LIN {X 0,Y 125.805,Z 374.565,A -85,B 0,C 180,E1 -26043.072,E2 -26043.072} C_VEL
LIN {X 0,Y 129.803,Z 368.331,A -85,B 0,C 180,E1 -26046.553,E2 -26046.553} C_VEL
LIN {X 0,Y 133.449,Z 362.382,A -85,B 0,C 180,E1 -26049.195,E2 -26049.195} C_VEL
LIN {X 0,Y 137.426,Z 355.46,A -85,B 0,C 180,E1 -26051.668,E2 -26051.668} C_VEL
LIN {X 0,Y 141.639,Z 347.287,A -85,B 0,C 180,E1 -26054,E2 -26054} C_VEL
LIN {X 0,Y 145.555,Z 338.782,A -85,B 0,C 180,E1 -26055.907,E2 -26055.907} C_VEL
LIN {X 0,Y 149.029,Z 330.073,A -85,B 0,C 180,E1 -26057.464,E2 -26057.464} C_VEL
LIN {X 0,Y 152.312,Z 320.32,A -85,B 0,C 180,E1 -26058.823,E2 -26058.823} C_VEL
LIN {X 0,Y 155.098,Z 310.244,A -85,B 0,C 180,E1 -26059.876,E2 -26059.876} C_VEL
LIN {X 0,Y 157.131,Z 300.522,A -85,B 0,C 180,E1 -26060.648,E2 -26060.648} C_VEL
LIN {X 0,Y 158.62,Z 290.465,A -85,B 0,C 180,E1 -26061.213,E2 -26061.213} C_VEL
LIN {X 0,Y 161.003,Z 261.314,A -85,B 0,C 180,E1 -26062.328,E2 -26062.328} C_VEL
LIN {X 0,Y 157.408,Z 250.953,A -85,B 0,C 180,E1 -26064.837,E2 -26064.837} C_VEL
LIN {X 0,Y 153.208,Z 240.952,A -85,B 0,C 180,E1 -26067.966,E2 -26067.966} C_VEL
LIN {X 0,Y 150.186,Z 234.641,A -85,B 0,C 180,E1 -26070.435,E2 -26070.435} C_VEL
LIN {X 0,Y 148.177,Z 231.492,A -85,B 0,C 180,E1 -26072.14,E2 -26072.14} C_VEL
LIN {X 0,Y 145.958,Z 229.192,A -85,B 0,C 180,E1 -26074.072,E2 -26074.072} C_VEL
LIN {X 0,Y 143.609,Z 228.041,A -85,B 0,C 180,E1 -26076.192,E2 -26076.192} C_VEL
LIN {X 0,Y 139.298,Z 226.814,A -85,B 0,C 180,E1 -26080.737,E2 -26080.737} C_VEL
LIN {X 0,Y 137.61,Z 225.498,A -85,B 0,C 180,E1 -26083.063,E2 -26083.063} C_VEL
LIN {X 0,Y 137.151,Z 224.801,A -85,B 0,C 180,E1 -26083.823,E2 -26083.823} C_VEL
LIN {X 0,Y 135.938,Z 222.42,A -85,B 0,C 180,E1 -26086.164,E2 -26086.164} C_VEL
LIN {X 0,Y 133.45,Z 219.624,A -85,B 0,C 180,E1 -26092.433,E2 -26092.433} C_VEL
LIN {X 0,Y 132.71,Z 217.42,A -85,B 0,C 180,E1 -26096.963,E2 -26096.963} C_VEL
LIN {X 0,Y 132.559,Z 216.943,A -85,B 0,C 180,E1 -26099.998,E2 -26099.998} C_VEL
LIN {X 0,Y 132.841,Z 217.769,A -85,B 0,C 180,E1 -26104.55,E2 -26104.55} C_VEL
LIN {X 0,Y 135.328,Z 222.024,A -85,B 0,C 180,E1 -26113.049,E2 -26113.049} C_VEL
LIN {X 0,Y 136.086,Z 222.758,A -85,B 0,C 180,E1 -26114.532,E2 -26114.532} C_VEL
LIN {X 0,Y 138.438,Z 226.502,A -85,B 0,C 180,E1 -26118.558,E2 -26118.558} C_VEL
LIN {X 0,Y 139.441,Z 227.752,A -85,B 0,C 180,E1 -26119.949,E2 -26119.949} C_VEL
LIN {X 0,Y 142.517,Z 232.304,A -85,B 0,C 180,E1 -26123.715,E2 -26123.715} C_VEL
LIN {X 0,Y 145.382,Z 236.828,A -85,B 0,C 180,E1 -26126.682,E2 -26126.682} C_VEL
LIN {X 0,Y 149.025,Z 242.882,A -85,B 0,C 180,E1 -26129.947,E2 -26129.947} C_VEL
LIN {X 0,Y 153.781,Z 251.654,A -85,B 0,C 180,E1 -26133.649,E2 -26133.649} C_VEL
LIN {X 0,Y 157.713,Z 259.969,A -85,B 0,C 180,E1 -26136.386,E2 -26136.386} C_VEL
LIN {X 0,Y 161.345,Z 269,A -85,B 0,C 180,E1 -26138.749,E2 -26138.749} C_VEL
LIN {X 0,Y 167.918,Z 287.949,A -85,B 0,C 180,E1 -26142.851,E2 -26142.851} C_VEL
LIN {X 0,Y 172.526,Z 300.417,A -85,B 0,C 180,E1 -26145.98,E2 -26145.98} C_VEL
LIN {X 0,Y 176.9,Z 310.843,A -85,B 0,C 180,E1 -26149.01,E2 -26149.01} C_VEL
LIN {X 0,Y 181.004,Z 319.354,A -85,B 0,C 180,E1 -26151.745,E2 -26151.745} C_VEL
LIN {X 0,Y 187.368,Z 329.918,A -85,B 0,C 180,E1 -26155.607,E2 -26155.607} C_VEL
LIN {X 0,Y 193.523,Z 338.128,A -85,B 0,C 180,E1 -26158.912,E2 -26158.912} C_VEL
LIN {X 0,Y 201.709,Z 346.752,A -85,B 0,C 180,E1 -26162.731,E2 -26162.731} C_VEL
LIN {X 0,Y 208.524,Z 352.554,A -85,B 0,C 180,E1 -26165.502,E2 -26165.502} C_VEL
LIN {X 0,Y 219.809,Z 360.018,A -85,B 0,C 180,E1 -26169.409,E2 -26169.409} C_VEL
LIN {X 0,Y 231.627,Z 366.133,A -85,B 0,C 180,E1 -26172.891,E2 -26172.891} C_VEL
LIN {X 0,Y 242.773,Z 371.001,A -85,B 0,C 180,E1 -26175.876,E2 -26175.876} C_VEL
LIN {X 0,Y 253.877,Z 375.462,A -85,B 0,C 180,E1 -26178.827,E2 -26178.827} C_VEL
LIN {X 0,Y 260.123,Z 378.03,A -85,B 0,C 180,E1 -26180.671,E2 -26180.671} C_VEL
LIN {X 0,Y 265.4,Z 380.136,A -85,B 0,C 180,E1 -26182.392,E2 -26182.392} C_VEL
LIN {X 0,Y 269.489,Z 381.819,A -85,B 0,C 180,E1 -26184.012,E2 -26184.012} C_VEL
LIN {X 0,Y 272.304,Z 383.12,A -85,B 0,C 180,E1 -26185.559,E2 -26185.559} C_VEL
LIN {X 0,Y 274.947,Z 384.042,A -85,B 0,C 180,E1 -26187.07,E2 -26187.07} C_VEL
LIN {X 0,Y 276.561,Z 384.593,A -85,B 0,C 180,E1 -26188.544,E2 -26188.544} C_VEL
LIN {X 0,Y 277.49,Z 384.769,A -85,B 0,C 180,E1 -26190,E2 -26190} C_VEL
LIN {X 0,Y 276.578,Z 384.592,A -85,B 0,C 180,E1 -26191.456,E2 -26191.456} C_VEL
LIN {X 0,Y 274.514,Z 383.905,A -85,B 0,C 180,E1 -26193.193,E2 -26193.193} C_VEL
LIN {X 0,Y 272.32,Z 383.12,A -85,B 0,C 180,E1 -26194.44,E2 -26194.44} C_VEL
LIN {X 0,Y 268.7,Z 381.499,A -85,B 0,C 180,E1 -26196.334,E2 -26196.334} C_VEL
LIN {X 0,Y 265.402,Z 380.136,A -85,B 0,C 180,E1 -26197.608,E2 -26197.608} C_VEL
LIN {X 0,Y 260.114,Z 378.03,A -85,B 0,C 180,E1 -26199.329,E2 -26199.329} C_VEL
LIN {X 0,Y 253.787,Z 375.464,A -85,B 0,C 180,E1 -26201.177,E2 -26201.177} C_VEL
LIN {X 0,Y 242.77,Z 371.007,A -85,B 0,C 180,E1 -26204.121,E2 -26204.121} C_VEL
LIN {X 0,Y 228.905,Z 364.849,A -85,B 0,C 180,E1 -26207.868,E2 -26207.868} C_VEL
LIN {X 0,Y 215.843,Z 357.681,A -85,B 0,C 180,E1 -26211.881,E2 -26211.881} C_VEL
LIN {X 0,Y 203.885,Z 348.801,A -85,B 0,C 180,E1 -26216.336,E2 -26216.336} C_VEL
LIN {X 0,Y 195.211,Z 340.03,A -85,B 0,C 180,E1 -26220.267,E2 -26220.267} C_VEL
LIN {X 0,Y 188.308,Z 331.272,A -85,B 0,C 180,E1 -26223.863,E2 -26223.863} C_VEL
LIN {X 0,Y 182.816,Z 322.622,A -85,B 0,C 180,E1 -26227.093,E2 -26227.093} C_VEL
LIN {X 0,Y 178.538,Z 314.413,A -85,B 0,C 180,E1 -26229.863,E2 -26229.863} C_VEL
LIN {X 0,Y 174.43,Z 305.201,A -85,B 0,C 180,E1 -26232.668,E2 -26232.668} C_VEL
LIN {X 0,Y 170.472,Z 295.07,A -85,B 0,C 180,E1 -26235.403,E2 -26235.403} C_VEL
LIN {X 0,Y 166.643,Z 284.283,A -85,B 0,C 180,E1 -26237.972,E2 -26237.972} C_VEL
LIN {X 0,Y 160.798,Z 267.492,A -85,B 0,C 180,E1 -26241.603,E2 -26241.603} C_VEL
LIN {X 0,Y 157.245,Z 258.936,A -85,B 0,C 180,E1 -26243.927,E2 -26243.927} C_VEL
LIN {X 0,Y 153.177,Z 250.497,A -85,B 0,C 180,E1 -26246.792,E2 -26246.792} C_VEL
LIN {X 0,Y 148.325,Z 241.59,A -85,B 0,C 180,E1 -26250.654,E2 -26250.654} C_VEL
LIN {X 0,Y 144.062,Z 234.686,A -85,B 0,C 180,E1 -26254.636,E2 -26254.636} C_VEL
LIN {X 0,Y 141.561,Z 230.897,A -85,B 0,C 180,E1 -26257.373,E2 -26257.373} C_VEL
LIN {X 0,Y 138.804,Z 226.859,A -85,B 0,C 180,E1 -26260.936,E2 -26260.936} C_VEL
LIN {X 0,Y 136.372,Z 223.381,A -85,B 0,C 180,E1 -26264.878,E2 -26264.878} C_VEL
LIN {X 0,Y 135.74,Z 222.313,A -85,B 0,C 180,E1 -26266.147,E2 -26266.147} C_VEL
LIN {X 0,Y 133.318,Z 219.298,A -85,B 0,C 180,E1 -26272.619,E2 -26272.619} C_VEL
LIN {X 0,Y 132.75,Z 217.516,A -85,B 0,C 180,E1 -26276.207,E2 -26276.207} C_VEL
LIN {X 0,Y 132.561,Z 216.929,A -85,B 0,C 180,E1 -26280.002,E2 -26280.002} C_VEL
LIN {X 0,Y 132.836,Z 217.812,A -85,B 0,C 180,E1 -26284.173,E2 -26284.173} C_VEL
LIN {X 0,Y 135.279,Z 221.975,A -85,B 0,C 180,E1 -26292.567,E2 -26292.567} C_VEL
LIN {X 0,Y 136.108,Z 222.806,A -85,B 0,C 180,E1 -26294.199,E2 -26294.199} C_VEL
LIN {X 0,Y 138.401,Z 226.445,A -85,B 0,C 180,E1 -26298.123,E2 -26298.123} C_VEL
LIN {X 0,Y 139.461,Z 227.805,A -85,B 0,C 180,E1 -26299.601,E2 -26299.601} C_VEL
LIN {X 0,Y 142.587,Z 232.444,A -85,B 0,C 180,E1 -26303.417,E2 -26303.417} C_VEL
LIN {X 0,Y 145.276,Z 236.637,A -85,B 0,C 180,E1 -26306.197,E2 -26306.197} C_VEL
LIN {X 0,Y 147.77,Z 240.777,A -85,B 0,C 180,E1 -26308.497,E2 -26308.497} C_VEL
LIN {X 0,Y 151.576,Z 249.615,A -85,B 0,C 180,E1 -26311.808,E2 -26311.808} C_VEL
LIN {X 0,Y 155.228,Z 259.333,A -85,B 0,C 180,E1 -26314.682,E2 -26314.682} C_VEL
LIN {X 0,Y 156.561,Z 263.582,A -85,B 0,C 180,E1 -26315.704,E2 -26315.704} C_VEL
LIN {X 0,Y 154.133,Z 291.552,A -85,B 0,C 180,E1 -26316.784,E2 -26316.784} C_VEL
LIN {X 0,Y 152.019,Z 304.342,A -85,B 0,C 180,E1 -26317.57,E2 -26317.57} C_VEL
LIN {X 0,Y 148.715,Z 317.11,A -85,B 0,C 180,E1 -26318.762,E2 -26318.762} C_VEL
LIN {X 0,Y 145.545,Z 326.619,A -85,B 0,C 180,E1 -26319.954,E2 -26319.954} C_VEL
LIN {X 0,Y 141.909,Z 335.89,A -85,B 0,C 180,E1 -26321.492,E2 -26321.492} C_VEL
LIN {X 0,Y 137.805,Z 344.829,A -85,B 0,C 180,E1 -26323.387,E2 -26323.387} C_VEL
LIN {X 0,Y 133.277,Z 353.35,A -85,B 0,C 180,E1 -26325.678,E2 -26325.678} C_VEL
LIN {X 0,Y 129.026,Z 360.564,A -85,B 0,C 180,E1 -26328.145,E2 -26328.145} C_VEL
LIN {X 0,Y 125.096,Z 366.763,A -85,B 0,C 180,E1 -26330.8,E2 -26330.8} C_VEL
LIN {X 0,Y 120.589,Z 373.298,A -85,B 0,C 180,E1 -26334.352,E2 -26334.352} C_VEL
LIN {X 0,Y 115.971,Z 379.719,A -85,B 0,C 180,E1 -26338.996,E2 -26338.996} C_VEL
LIN {X 0,Y 111.963,Z 384.849,A -85,B 0,C 180,E1 -26343.935,E2 -26343.935} C_VEL
LIN {X 0,Y 108.798,Z 388.838,A -85,B 0,C 180,E1 -26349.189,E2 -26349.189} C_VEL
LIN {X 0,Y 106.694,Z 391.797,A -85,B 0,C 180,E1 -26354.723,E2 -26354.723} C_VEL
LIN {X 0,Y 105.26,Z 394.259,A -85,B 0,C 180,E1 -26362.326,E2 -26362.326} C_VEL
LIN {X 0,Y 105.047,Z 394.855,A -85,B 0,C 180,E1 -26366.164,E2 -26366.164} C_VEL
LIN {X 0,Y 105.171,Z 395.017,A -85,B 0,C 180,E1 -26370,E2 -26370} C_VEL
LIN {X 0,Y 105.037,Z 394.855,A -85,B 0,C 180,E1 -26373.836,E2 -26373.836} C_VEL
LIN {X 0,Y 105.22,Z 394.258,A -85,B 0,C 180,E1 -26377.677,E2 -26377.677} C_VEL
LIN {X 0,Y 106.657,Z 391.796,A -85,B 0,C 180,E1 -26385.282,E2 -26385.282} C_VEL
LIN {X 0,Y 108.798,Z 388.838,A -85,B 0,C 180,E1 -26390.811,E2 -26390.811} C_VEL
LIN {X 0,Y 111.964,Z 384.849,A -85,B 0,C 180,E1 -26396.065,E2 -26396.065} C_VEL
LIN {X 0,Y 115.978,Z 379.719,A -85,B 0,C 180,E1 -26401.002,E2 -26401.002} C_VEL
LIN {X 0,Y 120.653,Z 373.3,A -85,B 0,C 180,E1 -26405.626,E2 -26405.626} C_VEL
LIN {X 0,Y 126.054,Z 365.38,A -85,B 0,C 180,E1 -26409.879,E2 -26409.879} C_VEL
LIN {X 0,Y 131.137,Z 357.186,A -85,B 0,C 180,E1 -26413.102,E2 -26413.102} C_VEL
LIN {X 0,Y 136.051,Z 348.229,A -85,B 0,C 180,E1 -26415.786,E2 -26415.786} C_VEL
LIN {X 0,Y 140.089,Z 339.94,A -85,B 0,C 180,E1 -26417.729,E2 -26417.729} C_VEL
LIN {X 0,Y 144.327,Z 329.881,A -85,B 0,C 180,E1 -26419.539,E2 -26419.539} C_VEL
LIN {X 0,Y 147.734,Z 320.128,A -85,B 0,C 180,E1 -26420.897,E2 -26420.897} C_VEL
LIN {X 0,Y 150.627,Z 310.053,A -85,B 0,C 180,E1 -26421.938,E2 -26421.938} C_VEL
LIN {X 0,Y 152.848,Z 299.656,A -85,B 0,C 180,E1 -26422.754,E2 -26422.754} C_VEL
LIN {X 0,Y 154.344,Z 289.518,A -85,B 0,C 180,E1 -26423.31,E2 -26423.31} C_VEL
LIN {X 0,Y 156.498,Z 263.378,A -85,B 0,C 180,E1 -26424.344,E2 -26424.344} C_VEL
LIN {X 0,Y 153.384,Z 254.234,A -85,B 0,C 180,E1 -26426.741,E2 -26426.741} C_VEL
LIN {X 0,Y 149.856,Z 245.431,A -85,B 0,C 180,E1 -26429.644,E2 -26429.644} C_VEL
LIN {X 0,Y 147.069,Z 239.541,A -85,B 0,C 180,E1 -26432.132,E2 -26432.132} C_VEL
LIN {X 0,Y 143.661,Z 234.104,A -85,B 0,C 180,E1 -26435.427,E2 -26435.427} C_VEL
LIN {X 0,Y 141.561,Z 230.911,A -85,B 0,C 180,E1 -26437.751,E2 -26437.751} C_VEL
LIN {X 0,Y 138.841,Z 226.876,A -85,B 0,C 180,E1 -26441.268,E2 -26441.268} C_VEL
LIN {X 0,Y 137.151,Z 224.801,A -85,B 0,C 180,E1 -26443.823,E2 -26443.823} C_VEL
LIN {X 0,Y 136.196,Z 224.118,A -85,B 0,C 180,E1 -26445.389,E2 -26445.389} C_VEL
LIN {X 0,Y 135.173,Z 224.623,A -85,B 0,C 180,E1 -26447.014,E2 -26447.014} C_VEL
LIN {X 0,Y 133.087,Z 226.856,A -85,B 0,C 180,E1 -26450.898,E2 -26450.898} C_VEL
LIN {X 0,Y 132.51,Z 226.72,A -85,B 0,C 180,E1 -26452.629,E2 -26452.629} C_VEL
LIN {X 0,Y 131.841,Z 224.506,A -85,B 0,C 180,E1 -26456.943,E2 -26456.943} C_VEL
LIN {X 0,Y 131.695,Z 223.98,A -85,B 0,C 180,E1 -26459.998,E2 -26459.998} C_VEL
LIN {X 0,Y 131.917,Z 224.797,A -85,B 0,C 180,E1 -26464.199,E2 -26464.199} C_VEL
LIN {X 0,Y 134.191,Z 228.935,A -85,B 0,C 180,E1 -26472.54,E2 -26472.54} C_VEL
LIN {X 0,Y 134.854,Z 229.744,A -85,B 0,C 180,E1 -26473.946,E2 -26473.946} C_VEL
LIN {X 0,Y 137.231,Z 233.475,A -85,B 0,C 180,E1 -26478.171,E2 -26478.171} C_VEL
LIN {X 0,Y 140.667,Z 238.788,A -85,B 0,C 180,E1 -26482.779,E2 -26482.779} C_VEL
LIN {X 0,Y 144.24,Z 244.672,A -85,B 0,C 180,E1 -26486.629,E2 -26486.629} C_VEL
LIN {X 0,Y 148.559,Z 252.715,A -85,B 0,C 180,E1 -26490.566,E2 -26490.566} C_VEL
LIN {X 0,Y 152.886,Z 261.619,A -85,B 0,C 180,E1 -26493.972,E2 -26493.972} C_VEL
LIN {X 0,Y 156.431,Z 270.321,A -85,B 0,C 180,E1 -26496.532,E2 -26496.532} C_VEL
LIN {X 0,Y 159.846,Z 280.417,A -85,B 0,C 180,E1 -26498.894,E2 -26498.894} C_VEL
LIN {X 0,Y 163.52,Z 292.327,A -85,B 0,C 180,E1 -26501.668,E2 -26501.668} C_VEL
LIN {X 0,Y 166.646,Z 301.839,A -85,B 0,C 180,E1 -26504.198,E2 -26504.198} C_VEL
LIN {X 0,Y 170.373,Z 312.012,A -85,B 0,C 180,E1 -26507.264,E2 -26507.264} C_VEL
LIN {X 0,Y 174.003,Z 320.511,A -85,B 0,C 180,E1 -26510.12,E2 -26510.12} C_VEL
LIN {X 0,Y 178.95,Z 329.727,A -85,B 0,C 180,E1 -26513.62,E2 -26513.62} C_VEL
LIN {X 0,Y 184.336,Z 337.842,A -85,B 0,C 180,E1 -26517.008,E2 -26517.008} C_VEL
LIN {X 0,Y 190.807,Z 345.637,A -85,B 0,C 180,E1 -26520.57,E2 -26520.57} C_VEL
LIN {X 0,Y 198.471,Z 352.947,A -85,B 0,C 180,E1 -26524.208,E2 -26524.208} C_VEL
LIN {X 0,Y 208.809,Z 360.329,A -85,B 0,C 180,E1 -26528.27,E2 -26528.27} C_VEL
LIN {X 0,Y 221.281,Z 367.038,A -85,B 0,C 180,E1 -26532.325,E2 -26532.325} C_VEL
LIN {X 0,Y 235.072,Z 372.796,A -85,B 0,C 180,E1 -26536.162,E2 -26536.162} C_VEL
LIN {X 0,Y 246.763,Z 377.026,A -85,B 0,C 180,E1 -26539.286,E2 -26539.286} C_VEL
LIN {X 0,Y 250.341,Z 378.294,A -85,B 0,C 180,E1 -26540.303,E2 -26540.303} C_VEL
LIN {X 0,Y 256.333,Z 380.383,A -85,B 0,C 180,E1 -26542.121,E2 -26542.121} C_VEL
LIN {X 0,Y 261.474,Z 382.187,A -85,B 0,C 180,E1 -26543.979,E2 -26543.979} C_VEL
LIN {X 0,Y 264.464,Z 383.33,A -85,B 0,C 180,E1 -26545.427,E2 -26545.427} C_VEL
LIN {X 0,Y 267.408,Z 384.296,A -85,B 0,C 180,E1 -26547.073,E2 -26547.073} C_VEL
LIN {X 0,Y 269.238,Z 384.79,A -85,B 0,C 180,E1 -26548.504,E2 -26548.504} C_VEL
LIN {X 0,Y 270.32,Z 384.959,A -85,B 0,C 180,E1 -26550,E2 -26550} C_VEL
LIN {X 0,Y 269.255,Z 384.789,A -85,B 0,C 180,E1 -26551.496,E2 -26551.496} C_VEL
LIN {X 0,Y 267.26,Z 384.252,A -85,B 0,C 180,E1 -26553.015,E2 -26553.015} C_VEL
LIN {X 0,Y 264.473,Z 383.33,A -85,B 0,C 180,E1 -26554.572,E2 -26554.572} C_VEL
LIN {X 0,Y 261.041,Z 382.05,A -85,B 0,C 180,E1 -26556.182,E2 -26556.182} C_VEL
LIN {X 0,Y 255.565,Z 380.133,A -85,B 0,C 180,E1 -26558.119,E2 -26558.119} C_VEL
LIN {X 0,Y 249.675,Z 378.08,A -85,B 0,C 180,E1 -26559.875,E2 -26559.875} C_VEL
LIN {X 0,Y 243.139,Z 375.755,A -85,B 0,C 180,E1 -26561.673,E2 -26561.673} C_VEL
LIN {X 0,Y 232.356,Z 371.724,A -85,B 0,C 180,E1 -26564.563,E2 -26564.563} C_VEL
LIN {X 0,Y 221.285,Z 367.03,A -85,B 0,C 180,E1 -26567.678,E2 -26567.678} C_VEL
LIN {X 0,Y 208.778,Z 360.329,A -85,B 0,C 180,E1 -26571.733,E2 -26571.733} C_VEL
LIN {X 0,Y 198.422,Z 352.928,A -85,B 0,C 180,E1 -26575.806,E2 -26575.806} C_VEL
LIN {X 0,Y 189.495,Z 344.213,A -85,B 0,C 180,E1 -26580.122,E2 -26580.122} C_VEL
LIN {X 0,Y 181.594,Z 333.93,A -85,B 0,C 180,E1 -26584.675,E2 -26584.675} C_VEL
LIN {X 0,Y 176.564,Z 325.504,A -85,B 0,C 180,E1 -26588.038,E2 -26588.038} C_VEL
LIN {X 0,Y 172.508,Z 317.015,A -85,B 0,C 180,E1 -26591.089,E2 -26591.089} C_VEL
LIN {X 0,Y 168.755,Z 307.716,A -85,B 0,C 180,E1 -26594.092,E2 -26594.092} C_VEL
LIN {X 0,Y 164.823,Z 296.331,A -85,B 0,C 180,E1 -26597.296,E2 -26597.296} C_VEL
LIN {X 0,Y 161.35,Z 285.284,A -85,B 0,C 180,E1 -26600.025,E2 -26600.025} C_VEL
LIN {X 0,Y 156.855,Z 271.534,A -85,B 0,C 180,E1 -26603.167,E2 -26603.167} C_VEL
LIN {X 0,Y 153.507,Z 263.119,A -85,B 0,C 180,E1 -26605.561,E2 -26605.561} C_VEL
LIN {X 0,Y 149.773,Z 255.115,A -85,B 0,C 180,E1 -26608.434,E2 -26608.434} C_VEL
LIN {X 0,Y 145.65,Z 247.223,A -85,B 0,C 180,E1 -26612.011,E2 -26612.011} C_VEL
LIN {X 0,Y 141.992,Z 240.935,A -85,B 0,C 180,E1 -26615.707,E2 -26615.707} C_VEL
LIN {X 0,Y 139.69,Z 237.263,A -85,B 0,C 180,E1 -26618.415,E2 -26618.415} C_VEL
LIN {X 0,Y 137.23,Z 233.485,A -85,B 0,C 180,E1 -26621.828,E2 -26621.828} C_VEL
LIN {X 0,Y 134.856,Z 229.733,A -85,B 0,C 180,E1 -26626.054,E2 -26626.054} C_VEL
LIN {X 0,Y 133.997,Z 228.754,A -85,B 0,C 180,E1 -26627.891,E2 -26627.891} C_VEL
LIN {X 0,Y 131.804,Z 224.426,A -85,B 0,C 180,E1 -26636.945,E2 -26636.945} C_VEL
LIN {X 0,Y 131.695,Z 223.98,A -85,B 0,C 180,E1 -26640.002,E2 -26640.002} C_VEL
LIN {X 0,Y 131.91,Z 224.849,A -85,B 0,C 180,E1 -26643.82,E2 -26643.82} C_VEL
LIN {X 0,Y 134.162,Z 228.904,A -85,B 0,C 180,E1 -26652.097,E2 -26652.097} C_VEL
LIN {X 0,Y 134.896,Z 229.829,A -85,B 0,C 180,E1 -26653.657,E2 -26653.657} C_VEL
LIN {X 0,Y 137.3,Z 233.518,A -85,B 0,C 180,E1 -26657.888,E2 -26657.888} C_VEL
LIN {X 0,Y 140.662,Z 238.815,A -85,B 0,C 180,E1 -26662.398,E2 -26662.398} C_VEL
LIN {X 0,Y 143.225,Z 243.038,A -85,B 0,C 180,E1 -26665.234,E2 -26665.234} C_VEL
LIN {X 0,Y 145.347,Z 246.893,A -85,B 0,C 180,E1 -26667.347,E2 -26667.347} C_VEL
LIN {X 0,Y 148.474,Z 254.677,A -85,B 0,C 180,E1 -26670.314,E2 -26670.314} C_VEL
LIN {X 0,Y 151.68,Z 263.756,A -85,B 0,C 180,E1 -26673.086,E2 -26673.086} C_VEL
LIN {X 0,Y 152.311,Z 265.891,A -85,B 0,C 180,E1 -26673.624,E2 -26673.624} C_VEL
LIN {X 0,Y 150.014,Z 291.057,A -85,B 0,C 180,E1 -26674.589,E2 -26674.589} C_VEL
LIN {X 0,Y 147.681,Z 304.729,A -85,B 0,C 180,E1 -26675.434,E2 -26675.434} C_VEL
LIN {X 0,Y 144.378,Z 316.918,A -85,B 0,C 180,E1 -26676.566,E2 -26676.566} C_VEL
LIN {X 0,Y 141.094,Z 326.427,A -85,B 0,C 180,E1 -26677.746,E2 -26677.746} C_VEL
LIN {X 0,Y 137.304,Z 335.698,A -85,B 0,C 180,E1 -26679.269,E2 -26679.269} C_VEL
LIN {X 0,Y 133.013,Z 344.637,A -85,B 0,C 180,E1 -26681.156,E2 -26681.156} C_VEL
LIN {X 0,Y 128.293,Z 353.159,A -85,B 0,C 180,E1 -26683.461,E2 -26683.461} C_VEL
LIN {X 0,Y 123.806,Z 360.371,A -85,B 0,C 180,E1 -26685.943,E2 -26685.943} C_VEL
LIN {X 0,Y 119.658,Z 366.571,A -85,B 0,C 180,E1 -26688.643,E2 -26688.643} C_VEL
LIN {X 0,Y 114.852,Z 373.105,A -85,B 0,C 180,E1 -26692.272,E2 -26692.272} C_VEL
LIN {X 0,Y 109.931,Z 379.527,A -85,B 0,C 180,E1 -26697.084,E2 -26697.084} C_VEL
LIN {X 0,Y 105.596,Z 384.656,A -85,B 0,C 180,E1 -26702.233,E2 -26702.233} C_VEL
LIN {X 0,Y 102.176,Z 388.646,A -85,B 0,C 180,E1 -26707.771,E2 -26707.771} C_VEL
LIN {X 0,Y 99.819,Z 391.604,A -85,B 0,C 180,E1 -26713.643,E2 -26713.643} C_VEL
LIN {X 0,Y 98.209,Z 394.066,A -85,B 0,C 180,E1 -26721.771,E2 -26721.771} C_VEL
LIN {X 0,Y 97.952,Z 394.663,A -85,B 0,C 180,E1 -26725.886,E2 -26725.886} C_VEL
LIN {X 0,Y 98.077,Z 394.825,A -85,B 0,C 180,E1 -26730,E2 -26730} C_VEL
LIN {X 0,Y 97.943,Z 394.663,A -85,B 0,C 180,E1 -26734.115,E2 -26734.115} C_VEL
LIN {X 0,Y 98.177,Z 394.066,A -85,B 0,C 180,E1 -26738.231,E2 -26738.231} C_VEL
LIN {X 0,Y 99.789,Z 391.603,A -85,B 0,C 180,E1 -26746.362,E2 -26746.362} C_VEL
LIN {X 0,Y 102.176,Z 388.646,A -85,B 0,C 180,E1 -26752.229,E2 -26752.229} C_VEL
LIN {X 0,Y 105.597,Z 384.656,A -85,B 0,C 180,E1 -26757.767,E2 -26757.767} C_VEL
LIN {X 0,Y 109.94,Z 379.527,A -85,B 0,C 180,E1 -26762.913,E2 -26762.913} C_VEL
LIN {X 0,Y 114.092,Z 374.211,A -85,B 0,C 180,E1 -26766.962,E2 -26766.962} C_VEL
LIN {X 0,Y 118.656,Z 367.946,A -85,B 0,C 180,E1 -26770.657,E2 -26770.657} C_VEL
LIN {X 0,Y 122.758,Z 361.998,A -85,B 0,C 180,E1 -26773.393,E2 -26773.393} C_VEL
LIN {X 0,Y 127.153,Z 355.076,A -85,B 0,C 180,E1 -26775.933,E2 -26775.933} C_VEL
LIN {X 0,Y 131.774,Z 346.903,A -85,B 0,C 180,E1 -26778.302,E2 -26778.302} C_VEL
LIN {X 0,Y 136.043,Z 338.398,A -85,B 0,C 180,E1 -26780.214,E2 -26780.214} C_VEL
LIN {X 0,Y 139.832,Z 329.69,A -85,B 0,C 180,E1 -26781.749,E2 -26781.749} C_VEL
LIN {X 0,Y 143.363,Z 319.936,A -85,B 0,C 180,E1 -26783.098,E2 -26783.098} C_VEL
LIN {X 0,Y 146.028,Z 311.149,A -85,B 0,C 180,E1 -26784.012,E2 -26784.012} C_VEL
LIN {X 0,Y 148.405,Z 300.83,A -85,B 0,C 180,E1 -26784.841,E2 -26784.841} C_VEL
LIN {X 0,Y 150.134,Z 290.04,A -85,B 0,C 180,E1 -26785.445,E2 -26785.445} C_VEL
LIN {X 0,Y 152.31,Z 265.897,A -85,B 0,C 180,E1 -26786.376,E2 -26786.376} C_VEL
LIN {X 0,Y 149.424,Z 257.228,A -85,B 0,C 180,E1 -26788.842,E2 -26788.842} C_VEL
LIN {X 0,Y 146.171,Z 248.781,A -85,B 0,C 180,E1 -26791.848,E2 -26791.848} C_VEL
LIN {X 0,Y 143.958,Z 244.179,A -85,B 0,C 180,E1 -26794.031,E2 -26794.031} C_VEL
LIN {X 0,Y 139.945,Z 237.56,A -85,B 0,C 180,E1 -26798.489,E2 -26798.489} C_VEL
LIN {X 0,Y 137.178,Z 233.405,A -85,B 0,C 180,E1 -26802.289,E2 -26802.289} C_VEL
LIN {X 0,Y 134.427,Z 229.087,A -85,B 0,C 180,E1 -26807.352,E2 -26807.352} C_VEL
LIN {X 0,Y 132.51,Z 226.72,A -85,B 0,C 180,E1 -26812.629,E2 -26812.629} C_VEL
LIN {X 0,Y 131.914,Z 226.312,A -85,B 0,C 180,E1 -26815.169,E2 -26815.169} C_VEL
LIN {X 0,Y 131.422,Z 227.189,A -85,B 0,C 180,E1 -26817.724,E2 -26817.724} C_VEL
LIN {X 0,Y 131.304,Z 233.102,A -85,B 0,C 180,E1 -26826.235,E2 -26826.235} C_VEL
LIN {X 0,Y 133.525,Z 236.461,A -85,B 0,C 180,E1 -26833.076,E2 -26833.076} C_VEL
LIN {X 0,Y 136.255,Z 241.002,A -85,B 0,C 180,E1 -26838.166,E2 -26838.166} C_VEL
LIN {X 0,Y 138.852,Z 245.312,A -85,B 0,C 180,E1 -26841.82,E2 -26841.82} C_VEL
LIN {X 0,Y 141.978,Z 250.739,A -85,B 0,C 180,E1 -26845.444,E2 -26845.444} C_VEL
LIN {X 0,Y 146.147,Z 258.956,A -85,B 0,C 180,E1 -26849.53,E2 -26849.53} C_VEL
LIN {X 0,Y 149.749,Z 266.936,A -85,B 0,C 180,E1 -26852.603,E2 -26852.603} C_VEL
LIN {X 0,Y 152.851,Z 275.032,A -85,B 0,C 180,E1 -26855.048,E2 -26855.048} C_VEL
LIN {X 0,Y 155.623,Z 283.893,A -85,B 0,C 180,E1 -26857.258,E2 -26857.258} C_VEL
LIN {X 0,Y 158.201,Z 293.431,A -85,B 0,C 180,E1 -26859.582,E2 -26859.582} C_VEL
LIN {X 0,Y 160.621,Z 302.077,A -85,B 0,C 180,E1 -26861.941,E2 -26861.941} C_VEL
LIN {X 0,Y 163.865,Z 312.37,A -85,B 0,C 180,E1 -26865.151,E2 -26865.151} C_VEL
LIN {X 0,Y 167.093,Z 321.102,A -85,B 0,C 180,E1 -26868.2,E2 -26868.2} C_VEL
LIN {X 0,Y 170.817,Z 329.404,A -85,B 0,C 180,E1 -26871.417,E2 -26871.417} C_VEL
LIN {X 0,Y 176.357,Z 338.883,A -85,B 0,C 180,E1 -26875.555,E2 -26875.555} C_VEL
LIN {X 0,Y 183.048,Z 347.523,A -85,B 0,C 180,E1 -26879.749,E2 -26879.749} C_VEL
LIN {X 0,Y 190.676,Z 355.012,A -85,B 0,C 180,E1 -26883.75,E2 -26883.75} C_VEL
LIN {X 0,Y 198.325,Z 360.784,A -85,B 0,C 180,E1 -26887.122,E2 -26887.122} C_VEL
LIN {X 0,Y 208.357,Z 366.557,A -85,B 0,C 180,E1 -26890.81,E2 -26890.81} C_VEL
LIN {X 0,Y 219.13,Z 371.396,A -85,B 0,C 180,E1 -26894.186,E2 -26894.186} C_VEL
LIN {X 0,Y 232.045,Z 376.059,A -85,B 0,C 180,E1 -26897.76,E2 -26897.76} C_VEL
LIN {X 0,Y 242.26,Z 379.271,A -85,B 0,C 180,E1 -26900.514,E2 -26900.514} C_VEL
LIN {X 0,Y 248.218,Z 381.101,A -85,B 0,C 180,E1 -26902.293,E2 -26902.293} C_VEL
LIN {X 0,Y 254.246,Z 382.894,A -85,B 0,C 180,E1 -26904.334,E2 -26904.334} C_VEL
LIN {X 0,Y 256.389,Z 383.547,A -85,B 0,C 180,E1 -26905.283,E2 -26905.283} C_VEL
LIN {X 0,Y 260.308,Z 384.659,A -85,B 0,C 180,E1 -26907.358,E2 -26907.358} C_VEL
LIN {X 0,Y 261.82,Z 384.989,A -85,B 0,C 180,E1 -26908.462,E2 -26908.462} C_VEL
LIN {X 0,Y 263.127,Z 385.15,A -85,B 0,C 180,E1 -26910,E2 -26910} C_VEL
LIN {X 0,Y 261.833,Z 384.989,A -85,B 0,C 180,E1 -26911.538,E2 -26911.538} C_VEL
LIN {X 0,Y 259.5,Z 384.463,A -85,B 0,C 180,E1 -26913.105,E2 -26913.105} C_VEL
LIN {X 0,Y 256.389,Z 383.547,A -85,B 0,C 180,E1 -26914.717,E2 -26914.717} C_VEL
LIN {X 0,Y 254.243,Z 382.9,A -85,B 0,C 180,E1 -26915.659,E2 -26915.659} C_VEL
LIN {X 0,Y 248.216,Z 381.105,A -85,B 0,C 180,E1 -26917.704,E2 -26917.704} C_VEL
LIN {X 0,Y 239.874,Z 378.574,A -85,B 0,C 180,E1 -26920.125,E2 -26920.125} C_VEL
LIN {X 0,Y 230.492,Z 375.541,A -85,B 0,C 180,E1 -26922.657,E2 -26922.657} C_VEL
LIN {X 0,Y 219.129,Z 371.397,A -85,B 0,C 180,E1 -26925.814,E2 -26925.814} C_VEL
LIN {X 0,Y 206.144,Z 365.462,A -85,B 0,C 180,E1 -26929.933,E2 -26929.933} C_VEL
LIN {X 0,Y 196.265,Z 359.356,A -85,B 0,C 180,E1 -26933.748,E2 -26933.748} C_VEL
LIN {X 0,Y 187.125,Z 351.786,A -85,B 0,C 180,E1 -26938.044,E2 -26938.044} C_VEL
LIN {X 0,Y 178.347,Z 341.68,A -85,B 0,C 180,E1 -26943.14,E2 -26943.14} C_VEL
LIN {X 0,Y 172.383,Z 332.311,A -85,B 0,C 180,E1 -26947.348,E2 -26947.348} C_VEL
LIN {X 0,Y 168.482,Z 324.438,A -85,B 0,C 180,E1 -26950.547,E2 -26950.547} C_VEL
LIN {X 0,Y 165.124,Z 315.895,A -85,B 0,C 180,E1 -26953.654,E2 -26953.654} C_VEL
LIN {X 0,Y 162.039,Z 306.645,A -85,B 0,C 180,E1 -26956.675,E2 -26956.675} C_VEL
LIN {X 0,Y 158.932,Z 296.166,A -85,B 0,C 180,E1 -26959.707,E2 -26959.707} C_VEL
LIN {X 0,Y 156.018,Z 285.27,A -85,B 0,C 180,E1 -26962.446,E2 -26962.446} C_VEL
LIN {X 0,Y 152.855,Z 274.991,A -85,B 0,C 180,E1 -26964.953,E2 -26964.953} C_VEL
LIN {X 0,Y 149.463,Z 266.215,A -85,B 0,C 180,E1 -26967.634,E2 -26967.634} C_VEL
LIN {X 0,Y 145.357,Z 257.39,A -85,B 0,C 180,E1 -26971.186,E2 -26971.186} C_VEL
LIN {X 0,Y 141.92,Z 250.624,A -85,B 0,C 180,E1 -26974.619,E2 -26974.619} C_VEL
LIN {X 0,Y 138.208,Z 244.087,A -85,B 0,C 180,E1 -26979.039,E2 -26979.039} C_VEL
LIN {X 0,Y 135.646,Z 240.035,A -85,B 0,C 180,E1 -26982.815,E2 -26982.815} C_VEL
LIN {X 0,Y 133.341,Z 236.033,A -85,B 0,C 180,E1 -26987.378,E2 -26987.378} C_VEL
LIN {X 0,Y 131.24,Z 232.9,A -85,B 0,C 180,E1 -26994.143,E2 -26994.143} C_VEL
LIN {X 0,Y 130.937,Z 231.499,A -85,B 0,C 180,E1 -26996.925,E2 -26996.925} C_VEL
LIN {X 0,Y 130.834,Z 231.137,A -85,B 0,C 180,E1 -27000.771,E2 -27000.771} C_VEL
LIN {X 0,Y 130.991,Z 231.876,A -85,B 0,C 180,E1 -27003.462,E2 -27003.462} C_VEL
LIN {X 0,Y 133.166,Z 235.92,A -85,B 0,C 180,E1 -27011.867,E2 -27011.867} C_VEL
LIN {X 0,Y 133.62,Z 236.654,A -85,B 0,C 180,E1 -27012.919,E2 -27012.919} C_VEL
LIN {X 0,Y 136.283,Z 241.055,A -85,B 0,C 180,E1 -27017.831,E2 -27017.831} C_VEL
LIN {X 0,Y 138.829,Z 245.276,A -85,B 0,C 180,E1 -27021.411,E2 -27021.411} C_VEL
LIN {X 0,Y 141.761,Z 250.31,A -85,B 0,C 180,E1 -27024.827,E2 -27024.827} C_VEL
LIN {X 0,Y 143.97,Z 255.564,A -85,B 0,C 180,E1 -27027.212,E2 -27027.212} C_VEL
LIN {X 0,Y 147.258,Z 264.889,A -85,B 0,C 180,E1 -27030.471,E2 -27030.471} C_VEL
LIN {X 0,Y 148.275,Z 268.355,A -85,B 0,C 180,E1 -27031.443,E2 -27031.443} C_VEL
LIN {X 0,Y 146.008,Z 291.609,A -85,B 0,C 180,E1 -27032.333,E2 -27032.333} C_VEL
LIN {X 0,Y 143.414,Z 305.625,A -85,B 0,C 180,E1 -27033.22,E2 -27033.22} C_VEL
LIN {X 0,Y 139.934,Z 317.734,A -85,B 0,C 180,E1 -27034.356,E2 -27034.356} C_VEL
LIN {X 0,Y 136.194,Z 327.866,A -85,B 0,C 180,E1 -27035.636,E2 -27035.636} C_VEL
LIN {X 0,Y 132.276,Z 336.857,A -85,B 0,C 180,E1 -27037.159,E2 -27037.159} C_VEL
LIN {X 0,Y 127.819,Z 345.579,A -85,B 0,C 180,E1 -27039.046,E2 -27039.046} C_VEL
LIN {X 0,Y 123.517,Z 352.967,A -85,B 0,C 180,E1 -27041.07,E2 -27041.07} C_VEL
LIN {X 0,Y 118.798,Z 360.18,A -85,B 0,C 180,E1 -27043.557,E2 -27043.557} C_VEL
LIN {X 0,Y 114.396,Z 366.378,A -85,B 0,C 180,E1 -27046.279,E2 -27046.279} C_VEL
LIN {X 0,Y 109.296,Z 372.912,A -85,B 0,C 180,E1 -27049.983,E2 -27049.983} C_VEL
LIN {X 0,Y 105.702,Z 377.417,A -85,B 0,C 180,E1 -27053.245,E2 -27053.245} C_VEL
LIN {X 0,Y 100.753,Z 382.908,A -85,B 0,C 180,E1 -27058.456,E2 -27058.456} C_VEL
LIN {X 0,Y 96.755,Z 387.236,A -85,B 0,C 180,E1 -27064.163,E2 -27064.163} C_VEL
LIN {X 0,Y 94.578,Z 389.605,A -85,B 0,C 180,E1 -27068.189,E2 -27068.189} C_VEL
LIN {X 0,Y 92.994,Z 391.411,A -85,B 0,C 180,E1 -27072.404,E2 -27072.404} C_VEL
LIN {X 0,Y 91.163,Z 393.874,A -85,B 0,C 180,E1 -27081.131,E2 -27081.131} C_VEL
LIN {X 0,Y 90.88,Z 394.472,A -85,B 0,C 180,E1 -27085.565,E2 -27085.565} C_VEL
LIN {X 0,Y 90.976,Z 394.634,A -85,B 0,C 180,E1 -27090,E2 -27090} C_VEL
LIN {X 0,Y 90.872,Z 394.471,A -85,B 0,C 180,E1 -27094.436,E2 -27094.436} C_VEL
LIN {X 0,Y 91.137,Z 393.873,A -85,B 0,C 180,E1 -27098.872,E2 -27098.872} C_VEL
LIN {X 0,Y 92.969,Z 391.411,A -85,B 0,C 180,E1 -27107.6,E2 -27107.6} C_VEL
LIN {X 0,Y 95.603,Z 388.453,A -85,B 0,C 180,E1 -27113.848,E2 -27113.848} C_VEL
LIN {X 0,Y 99.326,Z 384.463,A -85,B 0,C 180,E1 -27119.689,E2 -27119.689} C_VEL
LIN {X 0,Y 104.017,Z 379.335,A -85,B 0,C 180,E1 -27125.051,E2 -27125.051} C_VEL
LIN {X 0,Y 109.36,Z 372.915,A -85,B 0,C 180,E1 -27129.989,E2 -27129.989} C_VEL
LIN {X 0,Y 115.484,Z 364.995,A -85,B 0,C 180,E1 -27134.415,E2 -27134.415} C_VEL
LIN {X 0,Y 121.14,Z 356.802,A -85,B 0,C 180,E1 -27137.705,E2 -27137.705} C_VEL
LIN {X 0,Y 126.546,Z 347.845,A -85,B 0,C 180,E1 -27140.405,E2 -27140.405} C_VEL
LIN {X 0,Y 130.959,Z 339.557,A -85,B 0,C 180,E1 -27142.332,E2 -27142.332} C_VEL
LIN {X 0,Y 135.549,Z 329.498,A -85,B 0,C 180,E1 -27144.108,E2 -27144.108} C_VEL
LIN {X 0,Y 139.218,Z 319.745,A -85,B 0,C 180,E1 -27145.435,E2 -27145.435} C_VEL
LIN {X 0,Y 141.98,Z 310.957,A -85,B 0,C 180,E1 -27146.326,E2 -27146.326} C_VEL
LIN {X 0,Y 144.527,Z 300.118,A -85,B 0,C 180,E1 -27147.183,E2 -27147.183} C_VEL
LIN {X 0,Y 146.127,Z 290.669,A -85,B 0,C 180,E1 -27147.697,E2 -27147.697} C_VEL
LIN {X 0,Y 148.27,Z 268.223,A -85,B 0,C 180,E1 -27148.572,E2 -27148.572} C_VEL
LIN {X 0,Y 144.868,Z 257.923,A -85,B 0,C 180,E1 -27151.868,E2 -27151.868} C_VEL
LIN {X 0,Y 142.295,Z 251.417,A -85,B 0,C 180,E1 -27154.589,E2 -27154.589} C_VEL
LIN {X 0,Y 139.316,Z 246.128,A -85,B 0,C 180,E1 -27157.975,E2 -27157.975} C_VEL
LIN {X 0,Y 137.599,Z 243.269,A -85,B 0,C 180,E1 -27160.22,E2 -27160.22} C_VEL
LIN {X 0,Y 135.506,Z 239.845,A -85,B 0,C 180,E1 -27163.424,E2 -27163.424} C_VEL
LIN {X 0,Y 133.185,Z 235.928,A -85,B 0,C 180,E1 -27168.091,E2 -27168.091} C_VEL
LIN {X 0,Y 131.165,Z 232.659,A -85,B 0,C 180,E1 -27175.003,E2 -27175.003} C_VEL
LIN {X 0,Y 130.906,Z 231.409,A -85,B 0,C 180,E1 -27177.691,E2 -27177.691} C_VEL
LIN {X 0,Y 130.831,Z 231.017,A -85,B 0,C 180,E1 -27179.998,E2 -27179.998} C_VEL
LIN {X 0,Y 131,Z 231.801,A -85,B 0,C 180,E1 -27183.844,E2 -27183.844} C_VEL
LIN {X 0,Y 131.304,Z 233.102,A -85,B 0,C 180,E1 -27186.235,E2 -27186.235} C_VEL
LIN {X 0,Y 131.776,Z 235.02,A -85,B 0,C 180,E1 -27188.661,E2 -27188.661} C_VEL
LIN {X 0,Y 132.682,Z 240.102,A -85,B 0,C 180,E1 -27192.331,E2 -27192.331} C_VEL
LIN {X 0,Y 134.358,Z 246.777,A -85,B 0,C 180,E1 -27196.585,E2 -27196.585} C_VEL
LIN {X 0,Y 135.204,Z 248.565,A -85,B 0,C 180,E1 -27198.068,E2 -27198.068} C_VEL
LIN {X 0,Y 136.95,Z 251.559,A -85,B 0,C 180,E1 -27200.653,E2 -27200.653} C_VEL
LIN {X 0,Y 139.698,Z 256.634,A -85,B 0,C 180,E1 -27204.125,E2 -27204.125} C_VEL
LIN {X 0,Y 143.43,Z 264.443,A -85,B 0,C 180,E1 -27208.118,E2 -27208.118} C_VEL
LIN {X 0,Y 146.77,Z 272.379,A -85,B 0,C 180,E1 -27211.232,E2 -27211.232} C_VEL
LIN {X 0,Y 149.624,Z 280.414,A -85,B 0,C 180,E1 -27213.698,E2 -27213.698} C_VEL
LIN {X 0,Y 152.572,Z 291.972,A -85,B 0,C 180,E1 -27216.681,E2 -27216.681} C_VEL
LIN {X 0,Y 154.944,Z 302.312,A -85,B 0,C 180,E1 -27219.549,E2 -27219.549} C_VEL
LIN {X 0,Y 157.684,Z 312.762,A -85,B 0,C 180,E1 -27222.907,E2 -27222.907} C_VEL
LIN {X 0,Y 159.877,Z 320.091,A -85,B 0,C 180,E1 -27225.495,E2 -27225.495} C_VEL
LIN {X 0,Y 163.198,Z 329.17,A -85,B 0,C 180,E1 -27229.099,E2 -27229.099} C_VEL
LIN {X 0,Y 167.378,Z 337.684,A -85,B 0,C 180,E1 -27232.917,E2 -27232.917} C_VEL
LIN {X 0,Y 171.738,Z 344.657,A -85,B 0,C 180,E1 -27236.334,E2 -27236.334} C_VEL
LIN {X 0,Y 177.846,Z 352.153,A -85,B 0,C 180,E1 -27240.384,E2 -27240.384} C_VEL
LIN {X 0,Y 186.208,Z 359.757,A -85,B 0,C 180,E1 -27244.932,E2 -27244.932} C_VEL
LIN {X 0,Y 195.642,Z 365.996,A -85,B 0,C 180,E1 -27249.062,E2 -27249.062} C_VEL
LIN {X 0,Y 206.013,Z 371.083,A -85,B 0,C 180,E1 -27252.781,E2 -27252.781} C_VEL
LIN {X 0,Y 217.144,Z 375.273,A -85,B 0,C 180,E1 -27256.155,E2 -27256.155} C_VEL
LIN {X 0,Y 228.898,Z 378.87,A -85,B 0,C 180,E1 -27259.384,E2 -27259.384} C_VEL
LIN {X 0,Y 236.6,Z 380.921,A -85,B 0,C 180,E1 -27261.459,E2 -27261.459} C_VEL
LIN {X 0,Y 242.88,Z 382.545,A -85,B 0,C 180,E1 -27263.354,E2 -27263.354} C_VEL
LIN {X 0,Y 248.097,Z 383.77,A -85,B 0,C 180,E1 -27265.125,E2 -27265.125} C_VEL
LIN {X 0,Y 253.215,Z 384.979,A -85,B 0,C 180,E1 -27267.656,E2 -27267.656} C_VEL
LIN {X 0,Y 254.332,Z 385.19,A -85,B 0,C 180,E1 -27268.417,E2 -27268.417} C_VEL
LIN {X 0,Y 255.903,Z 385.341,A -85,B 0,C 180,E1 -27270,E2 -27270} C_VEL
LIN {X 0,Y 254.342,Z 385.19,A -85,B 0,C 180,E1 -27271.583,E2 -27271.583} C_VEL
LIN {X 0,Y 253.216,Z 384.979,A -85,B 0,C 180,E1 -27272.348,E2 -27272.348} C_VEL
LIN {X 0,Y 248.08,Z 383.77,A -85,B 0,C 180,E1 -27274.875,E2 -27274.875} C_VEL
LIN {X 0,Y 240.879,Z 382.04,A -85,B 0,C 180,E1 -27277.261,E2 -27277.261} C_VEL
LIN {X 0,Y 234.816,Z 380.485,A -85,B 0,C 180,E1 -27279.009,E2 -27279.009} C_VEL
LIN {X 0,Y 222.92,Z 377.152,A -85,B 0,C 180,E1 -27282.227,E2 -27282.227} C_VEL
LIN {X 0,Y 208.725,Z 372.214,A -85,B 0,C 180,E1 -27286.341,E2 -27286.341} C_VEL
LIN {X 0,Y 198.152,Z 367.368,A -85,B 0,C 180,E1 -27289.97,E2 -27289.97} C_VEL
LIN {X 0,Y 187.732,Z 360.932,A -85,B 0,C 180,E1 -27294.318,E2 -27294.318} C_VEL
LIN {X 0,Y 181.023,Z 355.296,A -85,B 0,C 180,E1 -27297.767,E2 -27297.767} C_VEL
LIN {X 0,Y 174.083,Z 347.68,A -85,B 0,C 180,E1 -27302.029,E2 -27302.029} C_VEL
LIN {X 0,Y 169.27,Z 340.835,A -85,B 0,C 180,E1 -27305.54,E2 -27305.54} C_VEL
LIN {X 0,Y 165.133,Z 333.402,A -85,B 0,C 180,E1 -27309.042,E2 -27309.042} C_VEL
LIN {X 0,Y 161.795,Z 325.436,A -85,B 0,C 180,E1 -27312.403,E2 -27312.403} C_VEL
LIN {X 0,Y 158.503,Z 315.662,A -85,B 0,C 180,E1 -27316.095,E2 -27316.095} C_VEL
LIN {X 0,Y 155.964,Z 306.325,A -85,B 0,C 180,E1 -27319.206,E2 -27319.206} C_VEL
LIN {X 0,Y 153.477,Z 296.004,A -85,B 0,C 180,E1 -27322.234,E2 -27322.234} C_VEL
LIN {X 0,Y 150.834,Z 284.56,A -85,B 0,C 180,E1 -27325.197,E2 -27325.197} C_VEL
LIN {X 0,Y 147.814,Z 275.062,A -85,B 0,C 180,E1 -27327.86,E2 -27327.86} C_VEL
LIN {X 0,Y 144.454,Z 266.774,A -85,B 0,C 180,E1 -27330.89,E2 -27330.89} C_VEL
LIN {X 0,Y 140.661,Z 258.608,A -85,B 0,C 180,E1 -27334.772,E2 -27334.772} C_VEL
LIN {X 0,Y 137.359,Z 252.272,A -85,B 0,C 180,E1 -27338.793,E2 -27338.793} C_VEL
LIN {X 0,Y 135.596,Z 249.222,A -85,B 0,C 180,E1 -27341.318,E2 -27341.318} C_VEL
LIN {X 0,Y 134.101,Z 246.548,A -85,B 0,C 180,E1 -27343.836,E2 -27343.836} C_VEL
LIN {X 0,Y 131.981,Z 242.757,A -85,B 0,C 180,E1 -27348.436,E2 -27348.436} C_VEL
LIN {X 0,Y 130.135,Z 239.1,A -85,B 0,C 180,E1 -27355.937,E2 -27355.937} C_VEL
LIN {X 0,Y 129.973,Z 238.292,A -85,B 0,C 180,E1 -27358.452,E2 -27358.452} C_VEL
LIN {X 0,Y 129.967,Z 238.197,A -85,B 0,C 180,E1 -27360.776,E2 -27360.776} C_VEL
LIN {X 0,Y 130.109,Z 239.067,A -85,B 0,C 180,E1 -27363.486,E2 -27363.486} C_VEL
LIN {X 0,Y 132.28,Z 243.289,A -85,B 0,C 180,E1 -27371.948,E2 -27371.948} C_VEL
LIN {X 0,Y 134.758,Z 247.716,A -85,B 0,C 180,E1 -27376.941,E2 -27376.941} C_VEL
LIN {X 0,Y 137.011,Z 251.663,A -85,B 0,C 180,E1 -27380.357,E2 -27380.357} C_VEL
LIN {X 0,Y 139.759,Z 256.799,A -85,B 0,C 180,E1 -27383.822,E2 -27383.822} C_VEL
LIN {X 0,Y 142.191,Z 263.462,A -85,B 0,C 180,E1 -27386.674,E2 -27386.674} C_VEL
LIN {X 0,Y 144.442,Z 270.716,A -85,B 0,C 180,E1 -27389.116,E2 -27389.116} C_VEL
LIN {X 0,Y 142.297,Z 291.693,A -85,B 0,C 180,E1 -27389.927,E2 -27389.927} C_VEL
LIN {X 0,Y 139.752,Z 305.044,A -85,B 0,C 180,E1 -27390.746,E2 -27390.746} C_VEL
LIN {X 0,Y 136.396,Z 316.535,A -85,B 0,C 180,E1 -27391.769,E2 -27391.769} C_VEL
LIN {X 0,Y 132.89,Z 326.045,A -85,B 0,C 180,E1 -27392.907,E2 -27392.907} C_VEL
LIN {X 0,Y 128.782,Z 335.315,A -85,B 0,C 180,E1 -27394.371,E2 -27394.371} C_VEL
LIN {X 0,Y 124.119,Z 344.254,A -85,B 0,C 180,E1 -27396.209,E2 -27396.209} C_VEL
LIN {X 0,Y 118.96,Z 352.775,A -85,B 0,C 180,E1 -27398.484,E2 -27398.484} C_VEL
LIN {X 0,Y 114.022,Z 359.988,A -85,B 0,C 180,E1 -27400.971,E2 -27400.971} C_VEL
LIN {X 0,Y 109.363,Z 366.186,A -85,B 0,C 180,E1 -27403.702,E2 -27403.702} C_VEL
LIN {X 0,Y 103.933,Z 372.72,A -85,B 0,C 180,E1 -27407.453,E2 -27407.453} C_VEL
LIN {X 0,Y 100.044,Z 377.224,A -85,B 0,C 180,E1 -27410.785,E2 -27410.785} C_VEL
LIN {X 0,Y 94.754,Z 382.716,A -85,B 0,C 180,E1 -27416.201,E2 -27416.201} C_VEL
LIN {X 0,Y 90.381,Z 387.043,A -85,B 0,C 180,E1 -27422.189,E2 -27422.189} C_VEL
LIN {X 0,Y 87.992,Z 389.413,A -85,B 0,C 180,E1 -27426.462,E2 -27426.462} C_VEL
LIN {X 0,Y 86.227,Z 391.219,A -85,B 0,C 180,E1 -27430.973,E2 -27430.973} C_VEL
LIN {X 0,Y 84.145,Z 393.682,A -85,B 0,C 180,E1 -27440.384,E2 -27440.384} C_VEL
LIN {X 0,Y 83.796,Z 394.28,A -85,B 0,C 180,E1 -27445.189,E2 -27445.189} C_VEL
LIN {X 0,Y 83.883,Z 394.442,A -85,B 0,C 180,E1 -27450,E2 -27450} C_VEL
LIN {X 0,Y 83.789,Z 394.28,A -85,B 0,C 180,E1 -27454.811,E2 -27454.811} C_VEL
LIN {X 0,Y 84.124,Z 393.682,A -85,B 0,C 180,E1 -27459.618,E2 -27459.618} C_VEL
LIN {X 0,Y 86.207,Z 391.219,A -85,B 0,C 180,E1 -27469.032,E2 -27469.032} C_VEL
LIN {X 0,Y 89.128,Z 388.261,A -85,B 0,C 180,E1 -27475.702,E2 -27475.702} C_VEL
LIN {X 0,Y 93.184,Z 384.27,A -85,B 0,C 180,E1 -27481.866,E2 -27481.866} C_VEL
LIN {X 0,Y 98.256,Z 379.142,A -85,B 0,C 180,E1 -27487.443,E2 -27487.443} C_VEL
LIN {X 0,Y 102.549,Z 374.397,A -85,B 0,C 180,E1 -27491.339,E2 -27491.339} C_VEL
LIN {X 0,Y 107.145,Z 368.937,A -85,B 0,C 180,E1 -27494.839,E2 -27494.839} C_VEL
LIN {X 0,Y 111.664,Z 363.24,A -85,B 0,C 180,E1 -27497.691,E2 -27497.691} C_VEL
LIN {X 0,Y 117.712,Z 354.693,A -85,B 0,C 180,E1 -27500.91,E2 -27500.91} C_VEL
LIN {X 0,Y 122.771,Z 346.519,A -85,B 0,C 180,E1 -27503.265,E2 -27503.265} C_VEL
LIN {X 0,Y 127.422,Z 338.015,A -85,B 0,C 180,E1 -27505.127,E2 -27505.127} C_VEL
LIN {X 0,Y 131.505,Z 329.306,A -85,B 0,C 180,E1 -27506.62,E2 -27506.62} C_VEL
LIN {X 0,Y 135.318,Z 319.553,A -85,B 0,C 180,E1 -27507.91,E2 -27507.91} C_VEL
LIN {X 0,Y 138.173,Z 310.766,A -85,B 0,C 180,E1 -27508.775,E2 -27508.775} C_VEL
LIN {X 0,Y 140.732,Z 300.341,A -85,B 0,C 180,E1 -27509.579,E2 -27509.579} C_VEL
LIN {X 0,Y 142.503,Z 290.008,A -85,B 0,C 180,E1 -27510.143,E2 -27510.143} C_VEL
LIN {X 0,Y 144.391,Z 270.562,A -85,B 0,C 180,E1 -27510.935,E2 -27510.935} C_VEL
LIN {X 0,Y 141.406,Z 261.171,A -85,B 0,C 180,E1 -27514.22,E2 -27514.22} C_VEL
LIN {X 0,Y 139.482,Z 256.222,A -85,B 0,C 180,E1 -27516.507,E2 -27516.507} C_VEL
LIN {X 0,Y 136.336,Z 250.33,A -85,B 0,C 180,E1 -27520.617,E2 -27520.617} C_VEL
LIN {X 0,Y 133.995,Z 246.393,A -85,B 0,C 180,E1 -27524.405,E2 -27524.405} C_VEL
LIN {X 0,Y 132.03,Z 242.815,A -85,B 0,C 180,E1 -27528.694,E2 -27528.694} C_VEL
LIN {X 0,Y 130.145,Z 239.256,A -85,B 0,C 180,E1 -27536.128,E2 -27536.128} C_VEL
LIN {X 0,Y 129.994,Z 238.311,A -85,B 0,C 180,E1 -27538.449,E2 -27538.449} C_VEL
LIN {X 0,Y 129.959,Z 238.168,A -85,B 0,C 180,E1 -27540.773,E2 -27540.773} C_VEL
LIN {X 0,Y 130.117,Z 239.007,A -85,B 0,C 180,E1 -27543.87,E2 -27543.87} C_VEL
LIN {X 0,Y 131.979,Z 242.769,A -85,B 0,C 180,E1 -27551.565,E2 -27551.565} C_VEL
LIN {X 0,Y 134.752,Z 247.666,A -85,B 0,C 180,E1 -27557.303,E2 -27557.303} C_VEL
LIN {X 0,Y 135.204,Z 248.565,A -85,B 0,C 180,E1 -27558.068,E2 -27558.068} C_VEL
LIN {X 0,Y 136.501,Z 251.561,A -85,B 0,C 180,E1 -27560.143,E2 -27560.143} C_VEL
LIN {X 0,Y 137.621,Z 255.508,A -85,B 0,C 180,E1 -27561.94,E2 -27561.94} C_VEL
LIN {X 0,Y 141.223,Z 270.959,A -85,B 0,C 180,E1 -27567.104,E2 -27567.104} C_VEL
LIN {X 0,Y 144.076,Z 278.379,A -85,B 0,C 180,E1 -27569.998,E2 -27569.998} C_VEL
LIN {X 0,Y 146.353,Z 286.023,A -85,B 0,C 180,E1 -27572.392,E2 -27572.392} C_VEL
LIN {X 0,Y 148.121,Z 294.497,A -85,B 0,C 180,E1 -27574.704,E2 -27574.704} C_VEL
LIN {X 0,Y 149.952,Z 304.168,A -85,B 0,C 180,E1 -27577.536,E2 -27577.536} C_VEL
LIN {X 0,Y 151.762,Z 312.883,A -85,B 0,C 180,E1 -27580.414,E2 -27580.414} C_VEL
LIN {X 0,Y 153.666,Z 320.808,A -85,B 0,C 180,E1 -27583.315,E2 -27583.315} C_VEL
LIN {X 0,Y 156.359,Z 329.781,A -85,B 0,C 180,E1 -27587.012,E2 -27587.012} C_VEL
LIN {X 0,Y 159.495,Z 337.636,A -85,B 0,C 180,E1 -27590.632,E2 -27590.632} C_VEL
LIN {X 0,Y 164.442,Z 346.557,A -85,B 0,C 180,E1 -27595.282,E2 -27595.282} C_VEL
LIN {X 0,Y 170.592,Z 354.497,A -85,B 0,C 180,E1 -27599.897,E2 -27599.897} C_VEL
LIN {X 0,Y 177.782,Z 361.221,A -85,B 0,C 180,E1 -27604.225,E2 -27604.225} C_VEL
LIN {X 0,Y 185.615,Z 366.651,A -85,B 0,C 180,E1 -27608.065,E2 -27608.065} C_VEL
LIN {X 0,Y 195.716,Z 371.805,A -85,B 0,C 180,E1 -27612.096,E2 -27612.096} C_VEL
LIN {X 0,Y 208.852,Z 376.696,A -85,B 0,C 180,E1 -27616.376,E2 -27616.376} C_VEL
LIN {X 0,Y 221.305,Z 380.183,A -85,B 0,C 180,E1 -27619.883,E2 -27619.883} C_VEL
LIN {X 0,Y 227.385,Z 381.591,A -85,B 0,C 180,E1 -27621.508,E2 -27621.508} C_VEL
LIN {X 0,Y 233.548,Z 382.927,A -85,B 0,C 180,E1 -27623.23,E2 -27623.23} C_VEL
LIN {X 0,Y 239.786,Z 384.168,A -85,B 0,C 180,E1 -27625.207,E2 -27625.207} C_VEL
LIN {X 0,Y 243.477,Z 384.899,A -85,B 0,C 180,E1 -27626.69,E2 -27626.69} C_VEL
LIN {X 0,Y 246.793,Z 385.393,A -85,B 0,C 180,E1 -27628.368,E2 -27628.368} C_VEL
LIN {X 0,Y 248.634,Z 385.533,A -85,B 0,C 180,E1 -27630,E2 -27630} C_VEL
LIN {X 0,Y 246.799,Z 385.393,A -85,B 0,C 180,E1 -27631.632,E2 -27631.632} C_VEL
LIN {X 0,Y 243.47,Z 384.899,A -85,B 0,C 180,E1 -27633.31,E2 -27633.31} C_VEL
LIN {X 0,Y 238.963,Z 384.015,A -85,B 0,C 180,E1 -27635.062,E2 -27635.062} C_VEL
LIN {X 0,Y 232.929,Z 382.817,A -85,B 0,C 180,E1 -27636.932,E2 -27636.932} C_VEL
LIN {X 0,Y 225.584,Z 381.222,A -85,B 0,C 180,E1 -27638.962,E2 -27638.962} C_VEL
LIN {X 0,Y 215.358,Z 378.626,A -85,B 0,C 180,E1 -27641.762,E2 -27641.762} C_VEL
LIN {X 0,Y 200.265,Z 373.772,A -85,B 0,C 180,E1 -27646.305,E2 -27646.305} C_VEL
LIN {X 0,Y 188.05,Z 368.064,A -85,B 0,C 180,E1 -27650.884,E2 -27650.884} C_VEL
LIN {X 0,Y 178.728,Z 361.993,A -85,B 0,C 180,E1 -27655.259,E2 -27655.259} C_VEL
LIN {X 0,Y 171.671,Z 355.576,A -85,B 0,C 180,E1 -27659.423,E2 -27659.423} C_VEL
LIN {X 0,Y 165.635,Z 348.296,A -85,B 0,C 180,E1 -27663.74,E2 -27663.74} C_VEL
LIN {X 0,Y 161.263,Z 341.095,A -85,B 0,C 180,E1 -27667.599,E2 -27667.599} C_VEL
LIN {X 0,Y 158.089,Z 334.374,A -85,B 0,C 180,E1 -27670.911,E2 -27670.911} C_VEL
LIN {X 0,Y 154.985,Z 325.452,A -85,B 0,C 180,E1 -27674.815,E2 -27674.815} C_VEL
LIN {X 0,Y 152.465,Z 315.924,A -85,B 0,C 180,E1 -27678.5,E2 -27678.5} C_VEL
LIN {X 0,Y 150.276,Z 305.856,A -85,B 0,C 180,E1 -27681.938,E2 -27681.938} C_VEL
LIN {X 0,Y 148.413,Z 296.103,A -85,B 0,C 180,E1 -27684.856,E2 -27684.856} C_VEL
LIN {X 0,Y 146.393,Z 286.049,A -85,B 0,C 180,E1 -27687.618,E2 -27687.618} C_VEL
LIN {X 0,Y 144.079,Z 278.353,A -85,B 0,C 180,E1 -27690.003,E2 -27690.003} C_VEL
LIN {X 0,Y 141.264,Z 271.115,A -85,B 0,C 180,E1 -27692.846,E2 -27692.846} C_VEL
LIN {X 0,Y 138.164,Z 264.012,A -85,B 0,C 180,E1 -27696.387,E2 -27696.387} C_VEL
LIN {X 0,Y 135.46,Z 258.473,A -85,B 0,C 180,E1 -27700.019,E2 -27700.019} C_VEL
LIN {X 0,Y 133.498,Z 254.819,A -85,B 0,C 180,E1 -27703.171,E2 -27703.171} C_VEL
LIN {X 0,Y 132.523,Z 252.999,A -85,B 0,C 180,E1 -27705.019,E2 -27705.019} C_VEL
LIN {X 0,Y 130.837,Z 249.625,A -85,B 0,C 180,E1 -27709.07,E2 -27709.07} C_VEL
LIN {X 0,Y 129.201,Z 246.05,A -85,B 0,C 180,E1 -27716.493,E2 -27716.493} C_VEL
LIN {X 0,Y 129.107,Z 245.352,A -85,B 0,C 180,E1 -27718.442,E2 -27718.442} C_VEL
LIN {X 0,Y 129.1,Z 245.261,A -85,B 0,C 180,E1 -27720.781,E2 -27720.781} C_VEL
LIN {X 0,Y 129.236,Z 246.426,A -85,B 0,C 180,E1 -27723.704,E2 -27723.704} C_VEL
LIN {X 0,Y 131.063,Z 250.077,A -85,B 0,C 180,E1 -27731.182,E2 -27731.182} C_VEL
LIN {X 0,Y 133.241,Z 254.305,A -85,B 0,C 180,E1 -27735.98,E2 -27735.98} C_VEL
LIN {X 0,Y 135.315,Z 258.195,A -85,B 0,C 180,E1 -27739.387,E2 -27739.387} C_VEL
LIN {X 0,Y 137.715,Z 263.078,A -85,B 0,C 180,E1 -27742.675,E2 -27742.675} C_VEL
LIN {X 0,Y 139.927,Z 270.197,A -85,B 0,C 180,E1 -27745.572,E2 -27745.572} C_VEL
LIN {X 0,Y 140.847,Z 273.345,A -85,B 0,C 180,E1 -27746.687,E2 -27746.687} C_VEL
LIN {X 0,Y 138.8,Z 292.233,A -85,B 0,C 180,E1 -27747.429,E2 -27747.429} C_VEL
LIN {X 0,Y 136.256,Z 304.852,A -85,B 0,C 180,E1 -27748.177,E2 -27748.177} C_VEL
LIN {X 0,Y 132.792,Z 316.343,A -85,B 0,C 180,E1 -27749.161,E2 -27749.161} C_VEL
LIN {X 0,Y 129.176,Z 325.853,A -85,B 0,C 180,E1 -27750.266,E2 -27750.266} C_VEL
LIN {X 0,Y 124.912,Z 335.123,A -85,B 0,C 180,E1 -27751.682,E2 -27751.682} C_VEL
LIN {X 0,Y 120.062,Z 344.062,A -85,B 0,C 180,E1 -27753.474,E2 -27753.474} C_VEL
LIN {X 0,Y 114.672,Z 352.583,A -85,B 0,C 180,E1 -27755.703,E2 -27755.703} C_VEL
LIN {X 0,Y 109.497,Z 359.796,A -85,B 0,C 180,E1 -27758.164,E2 -27758.164} C_VEL
LIN {X 0,Y 104.576,Z 365.994,A -85,B 0,C 180,E1 -27760.883,E2 -27760.883} C_VEL
LIN {X 0,Y 98.798,Z 372.527,A -85,B 0,C 180,E1 -27764.656,E2 -27764.656} C_VEL
LIN {X 0,Y 94.62,Z 377.031,A -85,B 0,C 180,E1 -27768.05,E2 -27768.05} C_VEL
LIN {X 0,Y 88.927,Z 382.524,A -85,B 0,C 180,E1 -27773.649,E2 -27773.649} C_VEL
LIN {X 0,Y 84.138,Z 386.851,A -85,B 0,C 180,E1 -27779.922,E2 -27779.922} C_VEL
LIN {X 0,Y 81.499,Z 389.22,A -85,B 0,C 180,E1 -27784.458,E2 -27784.458} C_VEL
LIN {X 0,Y 79.511,Z 391.026,A -85,B 0,C 180,E1 -27789.295,E2 -27789.295} C_VEL
LIN {X 0,Y 77.13,Z 393.49,A -85,B 0,C 180,E1 -27799.5,E2 -27799.5} C_VEL
LIN {X 0,Y 76.733,Z 394.089,A -85,B 0,C 180,E1 -27804.745,E2 -27804.745} C_VEL
LIN {X 0,Y 76.78,Z 394.251,A -85,B 0,C 180,E1 -27810,E2 -27810} C_VEL
LIN {X 0,Y 76.708,Z 394.088,A -85,B 0,C 180,E1 -27815.257,E2 -27815.257} C_VEL
LIN {X 0,Y 77.112,Z 393.49,A -85,B 0,C 180,E1 -27820.502,E2 -27820.502} C_VEL
LIN {X 0,Y 79.495,Z 391.026,A -85,B 0,C 180,E1 -27830.709,E2 -27830.709} C_VEL
LIN {X 0,Y 82.764,Z 388.069,A -85,B 0,C 180,E1 -27837.842,E2 -27837.842} C_VEL
LIN {X 0,Y 87.199,Z 384.077,A -85,B 0,C 180,E1 -27844.345,E2 -27844.345} C_VEL
LIN {X 0,Y 92.694,Z 378.949,A -85,B 0,C 180,E1 -27850.125,E2 -27850.125} C_VEL
LIN {X 0,Y 97.772,Z 373.687,A -85,B 0,C 180,E1 -27854.493,E2 -27854.493} C_VEL
LIN {X 0,Y 103.373,Z 367.369,A -85,B 0,C 180,E1 -27858.404,E2 -27858.404} C_VEL
LIN {X 0,Y 108.235,Z 361.422,A -85,B 0,C 180,E1 -27861.186,E2 -27861.186} C_VEL
LIN {X 0,Y 113.364,Z 354.501,A -85,B 0,C 180,E1 -27863.7,E2 -27863.7} C_VEL
LIN {X 0,Y 118.659,Z 346.327,A -85,B 0,C 180,E1 -27866.015,E2 -27866.015} C_VEL
LIN {X 0,Y 123.506,Z 337.824,A -85,B 0,C 180,E1 -27867.826,E2 -27867.826} C_VEL
LIN {X 0,Y 127.738,Z 329.115,A -85,B 0,C 180,E1 -27869.279,E2 -27869.279} C_VEL
LIN {X 0,Y 131.687,Z 319.362,A -85,B 0,C 180,E1 -27870.525,E2 -27870.525} C_VEL
LIN {X 0,Y 134.635,Z 310.575,A -85,B 0,C 180,E1 -27871.356,E2 -27871.356} C_VEL
LIN {X 0,Y 137.174,Z 300.647,A -85,B 0,C 180,E1 -27872.102,E2 -27872.102} C_VEL
LIN {X 0,Y 139.094,Z 289.919,A -85,B 0,C 180,E1 -27872.674,E2 -27872.674} C_VEL
LIN {X 0,Y 140.843,Z 273.382,A -85,B 0,C 180,E1 -27873.313,E2 -27873.313} C_VEL
LIN {X 0,Y 138.498,Z 265.45,A -85,B 0,C 180,E1 -27876.269,E2 -27876.269} C_VEL
LIN {X 0,Y 137.165,Z 261.867,A -85,B 0,C 180,E1 -27878.04,E2 -27878.04} C_VEL
LIN {X 0,Y 134.361,Z 256.342,A -85,B 0,C 180,E1 -27882.102,E2 -27882.102} C_VEL
LIN {X 0,Y 132.427,Z 252.821,A -85,B 0,C 180,E1 -27885.594,E2 -27885.594} C_VEL
LIN {X 0,Y 130.759,Z 249.553,A -85,B 0,C 180,E1 -27889.653,E2 -27889.653} C_VEL
LIN {X 0,Y 129.125,Z 245.397,A -85,B 0,C 180,E1 -27898.439,E2 -27898.439} C_VEL
LIN {X 0,Y 129.093,Z 245.22,A -85,B 0,C 180,E1 -27900.778,E2 -27900.778} C_VEL
LIN {X 0,Y 129.19,Z 245.939,A -85,B 0,C 180,E1 -27903.312,E2 -27903.312} C_VEL
LIN {X 0,Y 131.028,Z 250.004,A -85,B 0,C 180,E1 -27911.466,E2 -27911.466} C_VEL
LIN {X 0,Y 133.298,Z 254.4,A -85,B 0,C 180,E1 -27916.461,E2 -27916.461} C_VEL
LIN {X 0,Y 135.368,Z 258.302,A -85,B 0,C 180,E1 -27919.846,E2 -27919.846} C_VEL
LIN {X 0,Y 138.162,Z 264.026,A -85,B 0,C 180,E1 -27923.613,E2 -27923.613} C_VEL
LIN {X 0,Y 141.223,Z 270.959,A -85,B 0,C 180,E1 -27927.104,E2 -27927.104} C_VEL
LIN {X 0,Y 141.882,Z 274.256,A -85,B 0,C 180,E1 -27927.966,E2 -27927.966} C_VEL
LIN {X 0,Y 142.179,Z 280.607,A -85,B 0,C 180,E1 -27928.868,E2 -27928.868} C_VEL
LIN {X 0,Y 142.309,Z 286.976,A -85,B 0,C 180,E1 -27929.779,E2 -27929.779} C_VEL
LIN {X 0,Y 142.824,Z 290.303,A -85,B 0,C 180,E1 -27930.643,E2 -27930.643} C_VEL
LIN {X 0,Y 144.688,Z 302.772,A -85,B 0,C 180,E1 -27934.337,E2 -27934.337} C_VEL
LIN {X 0,Y 146.093,Z 312.456,A -85,B 0,C 180,E1 -27937.536,E2 -27937.536} C_VEL
LIN {X 0,Y 147.705,Z 321.225,A -85,B 0,C 180,E1 -27940.86,E2 -27940.86} C_VEL
LIN {X 0,Y 149.8,Z 330.303,A -85,B 0,C 180,E1 -27944.726,E2 -27944.726} C_VEL
LIN {X 0,Y 152.614,Z 338.987,A -85,B 0,C 180,E1 -27948.917,E2 -27948.917} C_VEL
LIN {X 0,Y 156.363,Z 346.817,A -85,B 0,C 180,E1 -27953.204,E2 -27953.204} C_VEL
LIN {X 0,Y 161.216,Z 354.121,A -85,B 0,C 180,E1 -27957.638,E2 -27957.638} C_VEL
LIN {X 0,Y 167.162,Z 360.62,A -85,B 0,C 180,E1 -27961.991,E2 -27961.991} C_VEL
LIN {X 0,Y 174.344,Z 366.369,A -85,B 0,C 180,E1 -27966.228,E2 -27966.228} C_VEL
LIN {X 0,Y 181.327,Z 370.563,A -85,B 0,C 180,E1 -27969.585,E2 -27969.585} C_VEL
LIN {X 0,Y 190.742,Z 374.762,A -85,B 0,C 180,E1 -27973.328,E2 -27973.328} C_VEL
LIN {X 0,Y 205.757,Z 379.494,A -85,B 0,C 180,E1 -27978.174,E2 -27978.174} C_VEL
LIN {X 0,Y 214.26,Z 381.532,A -85,B 0,C 180,E1 -27980.561,E2 -27980.561} C_VEL
LIN {X 0,Y 222.382,Z 383.106,A -85,B 0,C 180,E1 -27982.738,E2 -27982.738} C_VEL
LIN {X 0,Y 229.346,Z 384.273,A -85,B 0,C 180,E1 -27984.725,E2 -27984.725} C_VEL
LIN {X 0,Y 232.568,Z 384.795,A -85,B 0,C 180,E1 -27985.722,E2 -27985.722} C_VEL
LIN {X 0,Y 234.912,Z 385.132,A -85,B 0,C 180,E1 -27986.57,E2 -27986.57} C_VEL
LIN {X 0,Y 239.044,Z 385.619,A -85,B 0,C 180,E1 -27988.372,E2 -27988.372} C_VEL
LIN {X 0,Y 241.28,Z 385.728,A -85,B 0,C 180,E1 -27990,E2 -27990} C_VEL
LIN {X 0,Y 238.924,Z 385.604,A -85,B 0,C 180,E1 -27991.686,E2 -27991.686} C_VEL
LIN {X 0,Y 234.905,Z 385.132,A -85,B 0,C 180,E1 -27993.43,E2 -27993.43} C_VEL
LIN {X 0,Y 232.567,Z 384.797,A -85,B 0,C 180,E1 -27994.275,E2 -27994.275} C_VEL
LIN {X 0,Y 226.206,Z 383.804,A -85,B 0,C 180,E1 -27996.18,E2 -27996.18} C_VEL
LIN {X 0,Y 219.951,Z 382.652,A -85,B 0,C 180,E1 -27997.901,E2 -27997.901} C_VEL
LIN {X 0,Y 207.789,Z 380.008,A -85,B 0,C 180,E1 -28001.235,E2 -28001.235} C_VEL
LIN {X 0,Y 196.212,Z 376.721,A -85,B 0,C 180,E1 -28004.744,E2 -28004.744} C_VEL
LIN {X 0,Y 185.449,Z 372.528,A -85,B 0,C 180,E1 -28008.665,E2 -28008.665} C_VEL
LIN {X 0,Y 175.682,Z 367.266,A -85,B 0,C 180,E1 -28013.064,E2 -28013.064} C_VEL
LIN {X 0,Y 168.161,Z 361.504,A -85,B 0,C 180,E1 -28017.369,E2 -28017.369} C_VEL
LIN {X 0,Y 162.656,Z 355.85,A -85,B 0,C 180,E1 -28021.231,E2 -28021.231} C_VEL
LIN {X 0,Y 157.792,Z 349.224,A -85,B 0,C 180,E1 -28025.381,E2 -28025.381} C_VEL
LIN {X 0,Y 153.621,Z 341.353,A -85,B 0,C 180,E1 -28029.827,E2 -28029.827} C_VEL
LIN {X 0,Y 151.301,Z 335.188,A -85,B 0,C 180,E1 -28032.983,E2 -28032.983} C_VEL
LIN {X 0,Y 148.456,Z 324.996,A -85,B 0,C 180,E1 -28037.598,E2 -28037.598} C_VEL
LIN {X 0,Y 146.791,Z 316.398,A -85,B 0,C 180,E1 -28041.004,E2 -28041.004} C_VEL
LIN {X 0,Y 145.201,Z 306.428,A -85,B 0,C 180,E1 -28044.494,E2 -28044.494} C_VEL
LIN {X 0,Y 143.771,Z 296.329,A -85,B 0,C 180,E1 -28047.577,E2 -28047.577} C_VEL
LIN {X 0,Y 142.148,Z 287.359,A -85,B 0,C 180,E1 -28050.269,E2 -28050.269} C_VEL
LIN {X 0,Y 139.795,Z 279.495,A -85,B 0,C 180,E1 -28053.1,E2 -28053.1} C_VEL
LIN {X 0,Y 136.603,Z 271.351,A -85,B 0,C 180,E1 -28056.955,E2 -28056.955} C_VEL
LIN {X 0,Y 134,Z 265.406,A -85,B 0,C 180,E1 -28060.69,E2 -28060.69} C_VEL
LIN {X 0,Y 132.185,Z 261.769,A -85,B 0,C 180,E1 -28063.793,E2 -28063.793} C_VEL
LIN {X 0,Y 131.041,Z 259.461,A -85,B 0,C 180,E1 -28066.156,E2 -28066.156} C_VEL
LIN {X 0,Y 129.57,Z 256.358,A -85,B 0,C 180,E1 -28070.113,E2 -28070.113} C_VEL
LIN {X 0,Y 128.239,Z 252.421,A -85,B 0,C 180,E1 -28078.432,E2 -28078.432} C_VEL
LIN {X 0,Y 128.232,Z 252.332,A -85,B 0,C 180,E1 -28080.787,E2 -28080.787} C_VEL
LIN {X 0,Y 129.868,Z 256.877,A -85,B 0,C 180,E1 -28090.402,E2 -28090.402} C_VEL
LIN {X 0,Y 131.8,Z 260.959,A -85,B 0,C 180,E1 -28095.069,E2 -28095.069} C_VEL
LIN {X 0,Y 133.492,Z 264.372,A -85,B 0,C 180,E1 -28098.118,E2 -28098.118} C_VEL
LIN {X 0,Y 135.564,Z 269.074,A -85,B 0,C 180,E1 -28101.28,E2 -28101.28} C_VEL
LIN {X 0,Y 137.504,Z 276.092,A -85,B 0,C 180,E1 -28104.137,E2 -28104.137} C_VEL
LIN {X 0,Y 135.545,Z 292.962,A -85,B 0,C 180,E1 -28104.807,E2 -28104.807} C_VEL
LIN {X 0,Y 132.505,Z 306.521,A -85,B 0,C 180,E1 -28105.623,E2 -28105.623} C_VEL
LIN {X 0,Y 129.119,Z 317.159,A -85,B 0,C 180,E1 -28106.532,E2 -28106.532} C_VEL
LIN {X 0,Y 125.006,Z 327.293,A -85,B 0,C 180,E1 -28107.69,E2 -28107.69} C_VEL
LIN {X 0,Y 120.596,Z 336.281,A -85,B 0,C 180,E1 -28109.056,E2 -28109.056} C_VEL
LIN {X 0,Y 115.59,Z 345.004,A -85,B 0,C 180,E1 -28110.817,E2 -28110.817} C_VEL
LIN {X 0,Y 110.677,Z 352.391,A -85,B 0,C 180,E1 -28112.715,E2 -28112.715} C_VEL
LIN {X 0,Y 105.245,Z 359.604,A -85,B 0,C 180,E1 -28115.113,E2 -28115.113} C_VEL
LIN {X 0,Y 100.052,Z 365.801,A -85,B 0,C 180,E1 -28117.793,E2 -28117.793} C_VEL
LIN {X 0,Y 93.927,Z 372.335,A -85,B 0,C 180,E1 -28121.563,E2 -28121.563} C_VEL
LIN {X 0,Y 88.21,Z 377.937,A -85,B 0,C 180,E1 -28126.035,E2 -28126.035} C_VEL
LIN {X 0,Y 83.303,Z 382.332,A -85,B 0,C 180,E1 -28130.747,E2 -28130.747} C_VEL
LIN {X 0,Y 78.052,Z 386.658,A -85,B 0,C 180,E1 -28137.3,E2 -28137.3} C_VEL
LIN {X 0,Y 75.128,Z 389.028,A -85,B 0,C 180,E1 -28142.113,E2 -28142.113} C_VEL
LIN {X 0,Y 72.884,Z 390.834,A -85,B 0,C 180,E1 -28147.312,E2 -28147.312} C_VEL
LIN {X 0,Y 70.149,Z 393.298,A -85,B 0,C 180,E1 -28158.441,E2 -28158.441} C_VEL
LIN {X 0,Y 69.645,Z 393.896,A -85,B 0,C 180,E1 -28164.208,E2 -28164.208} C_VEL
LIN {X 0,Y 69.677,Z 394.059,A -85,B 0,C 180,E1 -28170,E2 -28170} C_VEL
LIN {X 0,Y 69.621,Z 393.896,A -85,B 0,C 180,E1 -28175.794,E2 -28175.794} C_VEL
LIN {X 0,Y 70.111,Z 393.297,A -85,B 0,C 180,E1 -28181.565,E2 -28181.565} C_VEL
LIN {X 0,Y 72.871,Z 390.834,A -85,B 0,C 180,E1 -28192.692,E2 -28192.692} C_VEL
LIN {X 0,Y 76.538,Z 387.876,A -85,B 0,C 180,E1 -28200.333,E2 -28200.333} C_VEL
LIN {X 0,Y 81.407,Z 383.885,A -85,B 0,C 180,E1 -28207.179,E2 -28207.179} C_VEL
LIN {X 0,Y 87.344,Z 378.756,A -85,B 0,C 180,E1 -28213.151,E2 -28213.151} C_VEL
LIN {X 0,Y 92.815,Z 373.494,A -85,B 0,C 180,E1 -28217.583,E2 -28217.583} C_VEL
LIN {X 0,Y 98.793,Z 367.177,A -85,B 0,C 180,E1 -28221.492,E2 -28221.492} C_VEL
LIN {X 0,Y 103.925,Z 361.23,A -85,B 0,C 180,E1 -28224.242,E2 -28224.242} C_VEL
LIN {X 0,Y 109.296,Z 354.309,A -85,B 0,C 180,E1 -28226.712,E2 -28226.712} C_VEL
LIN {X 0,Y 114.845,Z 346.136,A -85,B 0,C 180,E1 -28228.951,E2 -28228.951} C_VEL
LIN {X 0,Y 119.873,Z 337.632,A -85,B 0,C 180,E1 -28230.702,E2 -28230.702} C_VEL
LIN {X 0,Y 124.26,Z 328.923,A -85,B 0,C 180,E1 -28232.095,E2 -28232.095} C_VEL
LIN {X 0,Y 128.347,Z 319.171,A -85,B 0,C 180,E1 -28233.282,E2 -28233.282} C_VEL
LIN {X 0,Y 131.378,Z 310.383,A -85,B 0,C 180,E1 -28234.075,E2 -28234.075} C_VEL
LIN {X 0,Y 134.09,Z 299.984,A -85,B 0,C 180,E1 -28234.822,E2 -28234.822} C_VEL
LIN {X 0,Y 135.954,Z 289.972,A -85,B 0,C 180,E1 -28235.317,E2 -28235.317} C_VEL
LIN {X 0,Y 137.504,Z 276.093,A -85,B 0,C 180,E1 -28235.863,E2 -28235.863} C_VEL
LIN {X 0,Y 135.623,Z 269.275,A -85,B 0,C 180,E1 -28238.629,E2 -28238.629} C_VEL
LIN {X 0,Y 134.168,Z 265.722,A -85,B 0,C 180,E1 -28240.814,E2 -28240.814} C_VEL
LIN {X 0,Y 132.083,Z 261.552,A -85,B 0,C 180,E1 -28244.371,E2 -28244.371} C_VEL
LIN {X 0,Y 130.921,Z 259.219,A -85,B 0,C 180,E1 -28246.81,E2 -28246.81} C_VEL
LIN {X 0,Y 129.708,Z 256.476,A -85,B 0,C 180,E1 -28250.106,E2 -28250.106} C_VEL
LIN {X 0,Y 128.231,Z 252.333,A -85,B 0,C 180,E1 -28259.213,E2 -28259.213} C_VEL
LIN {X 0,Y 128.255,Z 252.488,A -85,B 0,C 180,E1 -28261.961,E2 -28261.961} C_VEL
LIN {X 0,Y 129.883,Z 256.967,A -85,B 0,C 180,E1 -28270.844,E2 -28270.844} C_VEL
LIN {X 0,Y 131.715,Z 260.771,A -85,B 0,C 180,E1 -28275.273,E2 -28275.273} C_VEL
LIN {X 0,Y 133.692,Z 264.822,A -85,B 0,C 180,E1 -28278.83,E2 -28278.83} C_VEL
LIN {X 0,Y 136.172,Z 270.323,A -85,B 0,C 180,E1 -28282.472,E2 -28282.472} C_VEL
LIN {X 0,Y 139.268,Z 278.068,A -85,B 0,C 180,E1 -28286.302,E2 -28286.302} C_VEL
LIN {X 0,Y 141.848,Z 286.215,A -85,B 0,C 180,E1 -28289.392,E2 -28289.392} C_VEL
LIN {X 0,Y 142.824,Z 290.303,A -85,B 0,C 180,E1 -28290.643,E2 -28290.643} C_VEL
LIN {X 0,Y 143.374,Z 293.43,A -85,B 0,C 180,E1 -28291.565,E2 -28291.565} C_VEL
LIN {X 0,Y 143.494,Z 296.88,A -85,B 0,C 180,E1 -28292.321,E2 -28292.321} C_VEL
LIN {X 0,Y 143.123,Z 302.346,A -85,B 0,C 180,E1 -28293.274,E2 -28293.274} C_VEL
LIN {X 0,Y 141.641,Z 313.171,A -85,B 0,C 180,E1 -28295.261,E2 -28295.261} C_VEL
LIN {X 0,Y 141.481,Z 317.178,A -85,B 0,C 180,E1 -28296.42,E2 -28296.42} C_VEL
LIN {X 0,Y 141.566,Z 317.901,A -85,B 0,C 180,E1 -28296.69,E2 -28296.69} C_VEL
LIN {X 0,Y 143.352,Z 329.703,A -85,B 0,C 180,E1 -28301.721,E2 -28301.721} C_VEL
LIN {X 0,Y 145.562,Z 339.134,A -85,B 0,C 180,E1 -28306.402,E2 -28306.402} C_VEL
LIN {X 0,Y 148.587,Z 347.08,A -85,B 0,C 180,E1 -28310.927,E2 -28310.927} C_VEL
LIN {X 0,Y 152.888,Z 354.771,A -85,B 0,C 180,E1 -28315.833,E2 -28315.833} C_VEL
LIN {X 0,Y 157.563,Z 360.556,A -85,B 0,C 180,E1 -28319.924,E2 -28319.924} C_VEL
LIN {X 0,Y 164.45,Z 366.656,A -85,B 0,C 180,E1 -28324.7,E2 -28324.7} C_VEL
LIN {X 0,Y 172.81,Z 371.942,A -85,B 0,C 180,E1 -28329.287,E2 -28329.287} C_VEL
LIN {X 0,Y 183.084,Z 376.413,A -85,B 0,C 180,E1 -28333.667,E2 -28333.667} C_VEL
LIN {X 0,Y 194.313,Z 379.908,A -85,B 0,C 180,E1 -28337.56,E2 -28337.56} C_VEL
LIN {X 0,Y 206.317,Z 382.555,A -85,B 0,C 180,E1 -28341.054,E2 -28341.054} C_VEL
LIN {X 0,Y 212.539,Z 383.65,A -85,B 0,C 180,E1 -28342.742,E2 -28342.742} C_VEL
LIN {X 0,Y 219.058,Z 384.548,A -85,B 0,C 180,E1 -28344.477,E2 -28344.477} C_VEL
LIN {X 0,Y 225.776,Z 385.38,A -85,B 0,C 180,E1 -28346.431,E2 -28346.431} C_VEL
LIN {X 0,Y 231.967,Z 385.903,A -85,B 0,C 180,E1 -28348.835,E2 -28348.835} C_VEL
LIN {X 0,Y 233.804,Z 385.926,A -85,B 0,C 180,E1 -28350,E2 -28350} C_VEL
LIN {X 0,Y 231.967,Z 385.903,A -85,B 0,C 180,E1 -28351.164,E2 -28351.164} C_VEL
LIN {X 0,Y 230.629,Z 385.827,A -85,B 0,C 180,E1 -28351.746,E2 -28351.746} C_VEL
LIN {X 0,Y 225.357,Z 385.341,A -85,B 0,C 180,E1 -28353.684,E2 -28353.684} C_VEL
LIN {X 0,Y 218.89,Z 384.538,A -85,B 0,C 180,E1 -28355.551,E2 -28355.551} C_VEL
LIN {X 0,Y 211.044,Z 383.415,A -85,B 0,C 180,E1 -28357.655,E2 -28357.655} C_VEL
LIN {X 0,Y 200.236,Z 381.344,A -85,B 0,C 180,E1 -28360.662,E2 -28360.662} C_VEL
LIN {X 0,Y 185.582,Z 377.333,A -85,B 0,C 180,E1 -28365.372,E2 -28365.372} C_VEL
LIN {X 0,Y 175.279,Z 373.155,A -85,B 0,C 180,E1 -28369.57,E2 -28369.57} C_VEL
LIN {X 0,Y 168.119,Z 369.283,A -85,B 0,C 180,E1 -28373.124,E2 -28373.124} C_VEL
LIN {X 0,Y 159.794,Z 362.743,A -85,B 0,C 180,E1 -28378.405,E2 -28378.405} C_VEL
LIN {X 0,Y 153.863,Z 356.123,A -85,B 0,C 180,E1 -28383.238,E2 -28383.238} C_VEL
LIN {X 0,Y 149.771,Z 349.487,A -85,B 0,C 180,E1 -28387.591,E2 -28387.591} C_VEL
LIN {X 0,Y 146.98,Z 343.294,A -85,B 0,C 180,E1 -28391.319,E2 -28391.319} C_VEL
LIN {X 0,Y 144.326,Z 334.286,A -85,B 0,C 180,E1 -28396.062,E2 -28396.062} C_VEL
LIN {X 0,Y 142.615,Z 325.446,A -85,B 0,C 180,E1 -28400.163,E2 -28400.163} C_VEL
LIN {X 0,Y 141.338,Z 315.85,A -85,B 0,C 180,E1 -28404.063,E2 -28404.063} C_VEL
LIN {X 0,Y 140.481,Z 307.324,A -85,B 0,C 180,E1 -28407.114,E2 -28407.114} C_VEL
LIN {X 0,Y 139.457,Z 296.631,A -85,B 0,C 180,E1 -28410.469,E2 -28410.469} C_VEL
LIN {X 0,Y 138.118,Z 288.725,A -85,B 0,C 180,E1 -28413.156,E2 -28413.156} C_VEL
LIN {X 0,Y 136.194,Z 282.089,A -85,B 0,C 180,E1 -28415.923,E2 -28415.923} C_VEL
LIN {X 0,Y 133.69,Z 275.292,A -85,B 0,C 180,E1 -28419.52,E2 -28419.52} C_VEL
LIN {X 0,Y 131.523,Z 270.013,A -85,B 0,C 180,E1 -28423.211,E2 -28423.211} C_VEL
LIN {X 0,Y 129.689,Z 266.061,A -85,B 0,C 180,E1 -28427.133,E2 -28427.133} C_VEL
LIN {X 0,Y 128.419,Z 263.14,A -85,B 0,C 180,E1 -28430.949,E2 -28430.949} C_VEL
LIN {X 0,Y 127.372,Z 259.482,A -85,B 0,C 180,E1 -28438.421,E2 -28438.421} C_VEL
LIN {X 0,Y 127.361,Z 259.366,A -85,B 0,C 180,E1 -28440.595,E2 -28440.595} C_VEL
LIN {X 0,Y 128.704,Z 263.694,A -85,B 0,C 180,E1 -28449.63,E2 -28449.63} C_VEL
LIN {X 0,Y 130.39,Z 267.597,A -85,B 0,C 180,E1 -28454.13,E2 -28454.13} C_VEL
LIN {X 0,Y 132.284,Z 271.785,A -85,B 0,C 180,E1 -28457.789,E2 -28457.789} C_VEL
LIN {X 0,Y 133.483,Z 274.997,A -85,B 0,C 180,E1 -28459.814,E2 -28459.814} C_VEL
LIN {X 0,Y 134.438,Z 278.921,A -85,B 0,C 180,E1 -28461.467,E2 -28461.467} C_VEL
LIN {X 0,Y 132.66,Z 293.209,A -85,B 0,C 180,E1 -28462.047,E2 -28462.047} C_VEL
LIN {X 0,Y 129.594,Z 306.329,A -85,B 0,C 180,E1 -28462.792,E2 -28462.792} C_VEL
LIN {X 0,Y 126.439,Z 316.091,A -85,B 0,C 180,E1 -28463.555,E2 -28463.555} C_VEL
LIN {X 0,Y 122.634,Z 325.47,A -85,B 0,C 180,E1 -28464.527,E2 -28464.527} C_VEL
LIN {X 0,Y 118.068,Z 334.739,A -85,B 0,C 180,E1 -28465.801,E2 -28465.801} C_VEL
LIN {X 0,Y 112.841,Z 343.678,A -85,B 0,C 180,E1 -28467.438,E2 -28467.438} C_VEL
LIN {X 0,Y 107.006,Z 352.2,A -85,B 0,C 180,E1 -28469.515,E2 -28469.515} C_VEL
LIN {X 0,Y 101.318,Z 359.412,A -85,B 0,C 180,E1 -28471.819,E2 -28471.819} C_VEL
LIN {X 0,Y 95.859,Z 365.609,A -85,B 0,C 180,E1 -28474.432,E2 -28474.432} C_VEL
LIN {X 0,Y 89.356,Z 372.143,A -85,B 0,C 180,E1 -28478.139,E2 -28478.139} C_VEL
LIN {X 0,Y 83.858,Z 377.211,A -85,B 0,C 180,E1 -28482.106,E2 -28482.106} C_VEL
LIN {X 0,Y 77.926,Z 382.14,A -85,B 0,C 180,E1 -28487.437,E2 -28487.437} C_VEL
LIN {X 0,Y 72.161,Z 386.466,A -85,B 0,C 180,E1 -28494.243,E2 -28494.243} C_VEL
LIN {X 0,Y 68.912,Z 388.835,A -85,B 0,C 180,E1 -28499.341,E2 -28499.341} C_VEL
LIN {X 0,Y 64.448,Z 392.038,A -85,B 0,C 180,E1 -28510.904,E2 -28510.904} C_VEL
LIN {X 0,Y 63.183,Z 393.106,A -85,B 0,C 180,E1 -28517.146,E2 -28517.146} C_VEL
LIN {X 0,Y 62.575,Z 393.704,A -85,B 0,C 180,E1 -28523.551,E2 -28523.551} C_VEL
LIN {X 0,Y 62.568,Z 393.867,A -85,B 0,C 180,E1 -28530,E2 -28530} C_VEL
LIN {X 0,Y 62.554,Z 393.704,A -85,B 0,C 180,E1 -28536.451,E2 -28536.451} C_VEL
LIN {X 0,Y 63.152,Z 393.105,A -85,B 0,C 180,E1 -28542.86,E2 -28542.86} C_VEL
LIN {X 0,Y 66.334,Z 390.641,A -85,B 0,C 180,E1 -28555.074,E2 -28555.074} C_VEL
LIN {X 0,Y 70.486,Z 387.684,A -85,B 0,C 180,E1 -28563.256,E2 -28563.256} C_VEL
LIN {X 0,Y 75.851,Z 383.692,A -85,B 0,C 180,E1 -28570.435,E2 -28570.435} C_VEL
LIN {X 0,Y 81.475,Z 379.263,A -85,B 0,C 180,E1 -28575.846,E2 -28575.846} C_VEL
LIN {X 0,Y 88.158,Z 373.3,A -85,B 0,C 180,E1 -28581.011,E2 -28581.011} C_VEL
LIN {X 0,Y 94.529,Z 366.985,A -85,B 0,C 180,E1 -28584.866,E2 -28584.866} C_VEL
LIN {X 0,Y 99.927,Z 361.037,A -85,B 0,C 180,E1 -28587.562,E2 -28587.562} C_VEL
LIN {X 0,Y 105.556,Z 354.117,A -85,B 0,C 180,E1 -28589.945,E2 -28589.945} C_VEL
LIN {X 0,Y 111.349,Z 345.944,A -85,B 0,C 180,E1 -28592.083,E2 -28592.083} C_VEL
LIN {X 0,Y 116.567,Z 337.44,A -85,B 0,C 180,E1 -28593.744,E2 -28593.744} C_VEL
LIN {X 0,Y 121.096,Z 328.731,A -85,B 0,C 180,E1 -28595.068,E2 -28595.068} C_VEL
LIN {X 0,Y 124.916,Z 320.052,A -85,B 0,C 180,E1 -28596.066,E2 -28596.066} C_VEL
LIN {X 0,Y 128.556,Z 309.786,A -85,B 0,C 180,E1 -28596.953,E2 -28596.953} C_VEL
LIN {X 0,Y 131.266,Z 299.638,A -85,B 0,C 180,E1 -28597.632,E2 -28597.632} C_VEL
LIN {X 0,Y 133.148,Z 289.781,A -85,B 0,C 180,E1 -28598.091,E2 -28598.091} C_VEL
LIN {X 0,Y 134.437,Z 278.927,A -85,B 0,C 180,E1 -28598.533,E2 -28598.533} C_VEL
LIN {X 0,Y 133.105,Z 273.787,A -85,B 0,C 180,E1 -28600.83,E2 -28600.83} C_VEL
LIN {X 0,Y 131.078,Z 269.034,A -85,B 0,C 180,E1 -28604.448,E2 -28604.448} C_VEL
LIN {X 0,Y 129.524,Z 265.711,A -85,B 0,C 180,E1 -28607.931,E2 -28607.931} C_VEL
LIN {X 0,Y 128.418,Z 263.108,A -85,B 0,C 180,E1 -28611.342,E2 -28611.342} C_VEL
LIN {X 0,Y 127.362,Z 259.418,A -85,B 0,C 180,E1 -28619.208,E2 -28619.208} C_VEL
LIN {X 0,Y 127.371,Z 259.492,A -85,B 0,C 180,E1 -28621.579,E2 -28621.579} C_VEL
LIN {X 0,Y 128.72,Z 263.796,A -85,B 0,C 180,E1 -28630.084,E2 -28630.084} C_VEL
LIN {X 0,Y 130.338,Z 267.457,A -85,B 0,C 180,E1 -28634.39,E2 -28634.39} C_VEL
LIN {X 0,Y 132.001,Z 271.154,A -85,B 0,C 180,E1 -28637.675,E2 -28637.675} C_VEL
LIN {X 0,Y 134.173,Z 276.484,A -85,B 0,C 180,E1 -28641.206,E2 -28641.206} C_VEL
LIN {X 0,Y 136.792,Z 284.043,A -85,B 0,C 180,E1 -28644.975,E2 -28644.975} C_VEL
LIN {X 0,Y 138.722,Z 291.468,A -85,B 0,C 180,E1 -28647.841,E2 -28647.841} C_VEL
LIN {X 0,Y 139.862,Z 300.035,A -85,B 0,C 180,E1 -28650.539,E2 -28650.539} C_VEL
LIN {X 0,Y 140.917,Z 311.3,A -85,B 0,C 180,E1 -28654.261,E2 -28654.261} C_VEL
LIN {X 0,Y 141.566,Z 317.901,A -85,B 0,C 180,E1 -28656.69,E2 -28656.69} C_VEL
LIN {X 0,Y 141.736,Z 322.38,A -85,B 0,C 180,E1 -28658.249,E2 -28658.249} C_VEL
LIN {X 0,Y 140.566,Z 330.293,A -85,B 0,C 180,E1 -28660.629,E2 -28660.629} C_VEL
LIN {X 0,Y 139.421,Z 337.814,A -85,B 0,C 180,E1 -28663.213,E2 -28663.213} C_VEL
LIN {X 0,Y 139.49,Z 341.634,A -85,B 0,C 180,E1 -28665.033,E2 -28665.033} C_VEL
LIN {X 0,Y 141.656,Z 348.681,A -85,B 0,C 180,E1 -28669.295,E2 -28669.295} C_VEL
LIN {X 0,Y 144.524,Z 354.704,A -85,B 0,C 180,E1 -28673.365,E2 -28673.365} C_VEL
LIN {X 0,Y 148.938,Z 361.086,A -85,B 0,C 180,E1 -28678.141,E2 -28678.141} C_VEL
LIN {X 0,Y 154.796,Z 366.94,A -85,B 0,C 180,E1 -28682.999,E2 -28682.999} C_VEL
LIN {X 0,Y 162.828,Z 372.459,A -85,B 0,C 180,E1 -28688.119,E2 -28688.119} C_VEL
LIN {X 0,Y 170.157,Z 376.049,A -85,B 0,C 180,E1 -28691.794,E2 -28691.794} C_VEL
LIN {X 0,Y 182.35,Z 380.128,A -85,B 0,C 180,E1 -28696.63,E2 -28696.63} C_VEL
LIN {X 0,Y 192.696,Z 382.546,A -85,B 0,C 180,E1 -28699.971,E2 -28699.971} C_VEL
LIN {X 0,Y 205.148,Z 384.53,A -85,B 0,C 180,E1 -28703.446,E2 -28703.446} C_VEL
LIN {X 0,Y 215.648,Z 385.656,A -85,B 0,C 180,E1 -28706.263,E2 -28706.263} C_VEL
LIN {X 0,Y 221.867,Z 386.063,A -85,B 0,C 180,E1 -28708.185,E2 -28708.185} C_VEL
LIN {X 0,Y 224.907,Z 386.143,A -85,B 0,C 180,E1 -28709.321,E2 -28709.321} C_VEL
LIN {X 0,Y 226.162,Z 386.128,A -85,B 0,C 180,E1 -28710,E2 -28710} C_VEL
LIN {X 0,Y 224.907,Z 386.143,A -85,B 0,C 180,E1 -28710.679,E2 -28710.679} C_VEL
LIN {X 0,Y 221.852,Z 386.063,A -85,B 0,C 180,E1 -28711.815,E2 -28711.815} C_VEL
LIN {X 0,Y 215.577,Z 385.658,A -85,B 0,C 180,E1 -28713.738,E2 -28713.738} C_VEL
LIN {X 0,Y 205.146,Z 384.534,A -85,B 0,C 180,E1 -28716.547,E2 -28716.547} C_VEL
LIN {X 0,Y 190.725,Z 382.177,A -85,B 0,C 180,E1 -28720.617,E2 -28720.617} C_VEL
LIN {X 0,Y 175.415,Z 378.05,A -85,B 0,C 180,E1 -28725.943,E2 -28725.943} C_VEL
LIN {X 0,Y 165.175,Z 373.755,A -85,B 0,C 180,E1 -28730.602,E2 -28730.602} C_VEL
LIN {X 0,Y 158.364,Z 369.706,A -85,B 0,C 180,E1 -28734.553,E2 -28734.553} C_VEL
LIN {X 0,Y 150.636,Z 362.968,A -85,B 0,C 180,E1 -28740.336,E2 -28740.336} C_VEL
LIN {X 0,Y 145.894,Z 356.921,A -85,B 0,C 180,E1 -28745.025,E2 -28745.025} C_VEL
LIN {X 0,Y 142.13,Z 349.751,A -85,B 0,C 180,E1 -28750.002,E2 -28750.002} C_VEL
LIN {X 0,Y 139.826,Z 342.871,A -85,B 0,C 180,E1 -28754.26,E2 -28754.26} C_VEL
LIN {X 0,Y 138.18,Z 334.921,A -85,B 0,C 180,E1 -28758.611,E2 -28758.611} C_VEL
LIN {X 0,Y 137.109,Z 325.784,A -85,B 0,C 180,E1 -28762.969,E2 -28762.969} C_VEL
LIN {X 0,Y 136.538,Z 317.218,A -85,B 0,C 180,E1 -28766.555,E2 -28766.555} C_VEL
LIN {X 0,Y 136.141,Z 308.199,A -85,B 0,C 180,E1 -28769.867,E2 -28769.867} C_VEL
LIN {X 0,Y 135.548,Z 298.107,A -85,B 0,C 180,E1 -28773.23,E2 -28773.23} C_VEL
LIN {X 0,Y 134.655,Z 291.745,A -85,B 0,C 180,E1 -28775.631,E2 -28775.631} C_VEL
LIN {X 0,Y 132.942,Z 285.04,A -85,B 0,C 180,E1 -28778.791,E2 -28778.791} C_VEL
LIN {X 0,Y 131.068,Z 279.418,A -85,B 0,C 180,E1 -28782.145,E2 -28782.145} C_VEL
LIN {X 0,Y 129.356,Z 275.038,A -85,B 0,C 180,E1 -28785.649,E2 -28785.649} C_VEL
LIN {X 0,Y 128.046,Z 271.945,A -85,B 0,C 180,E1 -28789.074,E2 -28789.074} C_VEL
LIN {X 0,Y 127.355,Z 270.02,A -85,B 0,C 180,E1 -28791.573,E2 -28791.573} C_VEL
LIN {X 0,Y 126.489,Z 266.428,A -85,B 0,C 180,E1 -28799.206,E2 -28799.206} C_VEL
LIN {X 0,Y 126.489,Z 266.469,A -85,B 0,C 180,E1 -28800.599,E2 -28800.599} C_VEL
LIN {X 0,Y 127.581,Z 270.573,A -85,B 0,C 180,E1 -28808.915,E2 -28808.915} C_VEL
LIN {X 0,Y 129.08,Z 274.379,A -85,B 0,C 180,E1 -28813.324,E2 -28813.324} C_VEL
LIN {X 0,Y 130.712,Z 278.439,A -85,B 0,C 180,E1 -28816.8,E2 -28816.8} C_VEL
LIN {X 0,Y 131.487,Z 280.968,A -85,B 0,C 180,E1 -28818.303,E2 -28818.303} C_VEL
LIN {X 0,Y 131.692,Z 281.92,A -85,B 0,C 180,E1 -28818.726,E2 -28818.726} C_VEL
LIN {X 0,Y 129.478,Z 296.262,A -85,B 0,C 180,E1 -28819.316,E2 -28819.316} C_VEL
LIN {X 0,Y 127.018,Z 306.138,A -85,B 0,C 180,E1 -28819.845,E2 -28819.845} C_VEL
LIN {X 0,Y 123.59,Z 316.363,A -85,B 0,C 180,E1 -28820.582,E2 -28820.582} C_VEL
LIN {X 0,Y 119.079,Z 326.91,A -85,B 0,C 180,E1 -28821.635,E2 -28821.635} C_VEL
LIN {X 0,Y 114.374,Z 335.898,A -85,B 0,C 180,E1 -28822.824,E2 -28822.824} C_VEL
LIN {X 0,Y 108.981,Z 344.62,A -85,B 0,C 180,E1 -28824.372,E2 -28824.372} C_VEL
LIN {X 0,Y 103.688,Z 352.008,A -85,B 0,C 180,E1 -28826.094,E2 -28826.094} C_VEL
LIN {X 0,Y 97.749,Z 359.22,A -85,B 0,C 180,E1 -28828.267,E2 -28828.267} C_VEL
LIN {X 0,Y 92.025,Z 365.418,A -85,B 0,C 180,E1 -28830.778,E2 -28830.778} C_VEL
LIN {X 0,Y 85.148,Z 371.951,A -85,B 0,C 180,E1 -28834.374,E2 -28834.374} C_VEL
LIN {X 0,Y 78.55,Z 377.554,A -85,B 0,C 180,E1 -28838.781,E2 -28838.781} C_VEL
LIN {X 0,Y 72.845,Z 381.948,A -85,B 0,C 180,E1 -28843.649,E2 -28843.649} C_VEL
LIN {X 0,Y 66.515,Z 386.274,A -85,B 0,C 180,E1 -28850.658,E2 -28850.658} C_VEL
LIN {X 0,Y 62.894,Z 388.643,A -85,B 0,C 180,E1 -28856.033,E2 -28856.033} C_VEL
LIN {X 0,Y 59.948,Z 390.448,A -85,B 0,C 180,E1 -28862.035,E2 -28862.035} C_VEL
LIN {X 0,Y 56.27,Z 392.914,A -85,B 0,C 180,E1 -28875.535,E2 -28875.535} C_VEL
LIN {X 0,Y 55.528,Z 393.513,A -85,B 0,C 180,E1 -28882.729,E2 -28882.729} C_VEL
LIN {X 0,Y 55.479,Z 393.676,A -85,B 0,C 180,E1 -28890,E2 -28890} C_VEL
LIN {X 0,Y 55.489,Z 393.512,A -85,B 0,C 180,E1 -28897.276,E2 -28897.276} C_VEL
LIN {X 0,Y 56.245,Z 392.913,A -85,B 0,C 180,E1 -28904.472,E2 -28904.472} C_VEL
LIN {X 0,Y 59.938,Z 390.448,A -85,B 0,C 180,E1 -28917.97,E2 -28917.97} C_VEL
LIN {X 0,Y 64.655,Z 387.492,A -85,B 0,C 180,E1 -28926.716,E2 -28926.716} C_VEL
LIN {X 0,Y 70.583,Z 383.5,A -85,B 0,C 180,E1 -28934.186,E2 -28934.186} C_VEL
LIN {X 0,Y 77.519,Z 378.384,A -85,B 0,C 180,E1 -28940.38,E2 -28940.38} C_VEL
LIN {X 0,Y 83.842,Z 373.107,A -85,B 0,C 180,E1 -28944.814,E2 -28944.814} C_VEL
LIN {X 0,Y 90.611,Z 366.792,A -85,B 0,C 180,E1 -28948.559,E2 -28948.559} C_VEL
LIN {X 0,Y 96.294,Z 360.845,A -85,B 0,C 180,E1 -28951.14,E2 -28951.14} C_VEL
LIN {X 0,Y 102.177,Z 353.924,A -85,B 0,C 180,E1 -28953.401,E2 -28953.401} C_VEL
LIN {X 0,Y 108.202,Z 345.752,A -85,B 0,C 180,E1 -28955.412,E2 -28955.412} C_VEL
LIN {X 0,Y 113.603,Z 337.249,A -85,B 0,C 180,E1 -28956.959,E2 -28956.959} C_VEL
LIN {X 0,Y 118.28,Z 328.54,A -85,B 0,C 180,E1 -28958.187,E2 -28958.187} C_VEL
LIN {X 0,Y 122.118,Z 320.09,A -85,B 0,C 180,E1 -28959.089,E2 -28959.089} C_VEL
LIN {X 0,Y 125.599,Z 310.723,A -85,B 0,C 180,E1 -28959.848,E2 -28959.848} C_VEL
LIN {X 0,Y 128.616,Z 299.967,A -85,B 0,C 180,E1 -28960.526,E2 -28960.526} C_VEL
LIN {X 0,Y 130.699,Z 289.431,A -85,B 0,C 180,E1 -28960.973,E2 -28960.973} C_VEL
LIN {X 0,Y 131.669,Z 281.815,A -85,B 0,C 180,E1 -28961.32,E2 -28961.32} C_VEL
LIN {X 0,Y 130.957,Z 279.119,A -85,B 0,C 180,E1 -28962.73,E2 -28962.73} C_VEL
LIN {X 0,Y 129.328,Z 275.011,A -85,B 0,C 180,E1 -28966.083,E2 -28966.083} C_VEL
LIN {X 0,Y 128.174,Z 272.217,A -85,B 0,C 180,E1 -28969.078,E2 -28969.078} C_VEL
LIN {X 0,Y 127.325,Z 269.965,A -85,B 0,C 180,E1 -28972.067,E2 -28972.067} C_VEL
LIN {X 0,Y 126.494,Z 266.337,A -85,B 0,C 180,E1 -28979.998,E2 -28979.998} C_VEL
LIN {X 0,Y 126.476,Z 266.877,A -85,B 0,C 180,E1 -28981.789,E2 -28981.789} C_VEL
LIN {X 0,Y 127.58,Z 270.623,A -85,B 0,C 180,E1 -28989.311,E2 -28989.311} C_VEL
LIN {X 0,Y 129.03,Z 274.262,A -85,B 0,C 180,E1 -28993.584,E2 -28993.584} C_VEL
LIN {X 0,Y 130.53,Z 277.933,A -85,B 0,C 180,E1 -28996.82,E2 -28996.82} C_VEL
LIN {X 0,Y 132.488,Z 283.62,A -85,B 0,C 180,E1 -29000.472,E2 -29000.472} C_VEL
LIN {X 0,Y 134.488,Z 290.845,A -85,B 0,C 180,E1 -29003.991,E2 -29003.991} C_VEL
LIN {X 0,Y 135.458,Z 297.213,A -85,B 0,C 180,E1 -29006.477,E2 -29006.477} C_VEL
LIN {X 0,Y 135.946,Z 304.381,A -85,B 0,C 180,E1 -29008.85,E2 -29008.85} C_VEL
LIN {X 0,Y 136.3,Z 312.789,A -85,B 0,C 180,E1 -29011.748,E2 -29011.748} C_VEL
LIN {X 0,Y 136.758,Z 321.92,A -85,B 0,C 180,E1 -29015.316,E2 -29015.316} C_VEL
LIN {X 0,Y 137.672,Z 331.438,A -85,B 0,C 180,E1 -29019.651,E2 -29019.651} C_VEL
LIN {X 0,Y 138.824,Z 338.515,A -85,B 0,C 180,E1 -29023.275,E2 -29023.275} C_VEL
LIN {X 0,Y 139.49,Z 341.634,A -85,B 0,C 180,E1 -29025.033,E2 -29025.033} C_VEL
LIN {X 0,Y 139.881,Z 345.389,A -85,B 0,C 180,E1 -29026.927,E2 -29026.927} C_VEL
LIN {X 0,Y 139.17,Z 351.928,A -85,B 0,C 180,E1 -29030.021,E2 -29030.021} C_VEL
LIN {X 0,Y 138.874,Z 357.801,A -85,B 0,C 180,E1 -29033.256,E2 -29033.256} C_VEL
LIN {X 0,Y 139.844,Z 360.628,A -85,B 0,C 180,E1 -29035.315,E2 -29035.315} C_VEL
LIN {X 0,Y 145.439,Z 367.22,A -85,B 0,C 180,E1 -29041.104,E2 -29041.104} C_VEL
LIN {X 0,Y 152.977,Z 372.902,A -85,B 0,C 180,E1 -29046.752,E2 -29046.752} C_VEL
LIN {X 0,Y 159.98,Z 376.591,A -85,B 0,C 180,E1 -29050.818,E2 -29050.818} C_VEL
LIN {X 0,Y 170.888,Z 380.44,A -85,B 0,C 180,E1 -29055.714,E2 -29055.714} C_VEL
LIN {X 0,Y 179.156,Z 382.52,A -85,B 0,C 180,E1 -29058.72,E2 -29058.72} C_VEL
LIN {X 0,Y 191.401,Z 384.611,A -85,B 0,C 180,E1 -29062.472,E2 -29062.472} C_VEL
LIN {X 0,Y 204.81,Z 385.951,A -85,B 0,C 180,E1 -29066.065,E2 -29066.065} C_VEL
LIN {X 0,Y 212.389,Z 386.318,A -85,B 0,C 180,E1 -29068.104,E2 -29068.104} C_VEL
LIN {X 0,Y 218.063,Z 386.343,A -85,B 0,C 180,E1 -29070,E2 -29070} C_VEL
LIN {X 0,Y 211.001,Z 386.259,A -85,B 0,C 180,E1 -29072.27,E2 -29072.27} C_VEL
LIN {X 0,Y 204.322,Z 385.913,A -85,B 0,C 180,E1 -29074.065,E2 -29074.065} C_VEL
LIN {X 0,Y 191.401,Z 384.612,A -85,B 0,C 180,E1 -29077.526,E2 -29077.526} C_VEL
LIN {X 0,Y 178.963,Z 382.5,A -85,B 0,C 180,E1 -29081.324,E2 -29081.324} C_VEL
LIN {X 0,Y 167.784,Z 379.549,A -85,B 0,C 180,E1 -29085.554,E2 -29085.554} C_VEL
LIN {X 0,Y 155.651,Z 374.492,A -85,B 0,C 180,E1 -29091.578,E2 -29091.578} C_VEL
LIN {X 0,Y 148.814,Z 370.056,A -85,B 0,C 180,E1 -29096.197,E2 -29096.197} C_VEL
LIN {X 0,Y 141.707,Z 363.15,A -85,B 0,C 180,E1 -29102.532,E2 -29102.532} C_VEL
LIN {X 0,Y 137.557,Z 356.658,A -85,B 0,C 180,E1 -29107.813,E2 -29107.813} C_VEL
LIN {X 0,Y 134.651,Z 349.42,A -85,B 0,C 180,E1 -29113.056,E2 -29113.056} C_VEL
LIN {X 0,Y 133.16,Z 342.116,A -85,B 0,C 180,E1 -29117.637,E2 -29117.637} C_VEL
LIN {X 0,Y 132.331,Z 334.93,A -85,B 0,C 180,E1 -29121.683,E2 -29121.683} C_VEL
LIN {X 0,Y 131.99,Z 326.27,A -85,B 0,C 180,E1 -29125.918,E2 -29125.918} C_VEL
LIN {X 0,Y 131.993,Z 316.313,A -85,B 0,C 180,E1 -29130.109,E2 -29130.109} C_VEL
LIN {X 0,Y 132.117,Z 306.499,A -85,B 0,C 180,E1 -29133.674,E2 -29133.674} C_VEL
LIN {X 0,Y 131.84,Z 298.652,A -85,B 0,C 180,E1 -29136.54,E2 -29136.54} C_VEL
LIN {X 0,Y 130.921,Z 292.512,A -85,B 0,C 180,E1 -29139.375,E2 -29139.375} C_VEL
LIN {X 0,Y 129.346,Z 285.906,A -85,B 0,C 180,E1 -29143.224,E2 -29143.224} C_VEL
LIN {X 0,Y 127.877,Z 281.398,A -85,B 0,C 180,E1 -29146.899,E2 -29146.899} C_VEL
LIN {X 0,Y 126.722,Z 278.293,A -85,B 0,C 180,E1 -29150.424,E2 -29150.424} C_VEL
LIN {X 0,Y 126.255,Z 276.853,A -85,B 0,C 180,E1 -29152.405,E2 -29152.405} C_VEL
LIN {X 0,Y 125.613,Z 273.566,A -85,B 0,C 180,E1 -29159.2,E2 -29159.2} C_VEL
LIN {X 0,Y 125.606,Z 273.616,A -85,B 0,C 180,E1 -29160.402,E2 -29160.402} C_VEL
LIN {X 0,Y 126.474,Z 277.486,A -85,B 0,C 180,E1 -29168.188,E2 -29168.188} C_VEL
LIN {X 0,Y 127.689,Z 280.876,A -85,B 0,C 180,E1 -29172.215,E2 -29172.215} C_VEL
LIN {X 0,Y 129.01,Z 284.719,A -85,B 0,C 180,E1 -29175.504,E2 -29175.504} C_VEL
LIN {X 0,Y 129.161,Z 285.199,A -85,B 0,C 180,E1 -29175.854,E2 -29175.854} C_VEL
LIN {X 0,Y 127.19,Z 296.568,A -85,B 0,C 180,E1 -29176.32,E2 -29176.32} C_VEL
LIN {X 0,Y 124.785,Z 305.947,A -85,B 0,C 180,E1 -29176.775,E2 -29176.775} C_VEL
LIN {X 0,Y 121.06,Z 316.708,A -85,B 0,C 180,E1 -29177.483,E2 -29177.483} C_VEL
LIN {X 0,Y 116.65,Z 326.718,A -85,B 0,C 180,E1 -29178.394,E2 -29178.394} C_VEL
LIN {X 0,Y 111.814,Z 335.707,A -85,B 0,C 180,E1 -29179.472,E2 -29179.472} C_VEL
LIN {X 0,Y 106.246,Z 344.428,A -85,B 0,C 180,E1 -29180.879,E2 -29180.879} C_VEL
LIN {X 0,Y 100.755,Z 351.815,A -85,B 0,C 180,E1 -29182.448,E2 -29182.448} C_VEL
LIN {X 0,Y 94.589,Z 359.028,A -85,B 0,C 180,E1 -29184.471,E2 -29184.471} C_VEL
LIN {X 0,Y 88.587,Z 365.225,A -85,B 0,C 180,E1 -29186.811,E2 -29186.811} C_VEL
LIN {X 0,Y 81.337,Z 371.758,A -85,B 0,C 180,E1 -29190.226,E2 -29190.226} C_VEL
LIN {X 0,Y 75.817,Z 376.26,A -85,B 0,C 180,E1 -29193.461,E2 -29193.461} C_VEL
LIN {X 0,Y 68.128,Z 381.756,A -85,B 0,C 180,E1 -29199.314,E2 -29199.314} C_VEL
LIN {X 0,Y 61.177,Z 386.082,A -85,B 0,C 180,E1 -29206.428,E2 -29206.428} C_VEL
LIN {X 0,Y 57.134,Z 388.451,A -85,B 0,C 180,E1 -29212.046,E2 -29212.046} C_VEL
LIN {X 0,Y 53.743,Z 390.255,A -85,B 0,C 180,E1 -29218.461,E2 -29218.461} C_VEL
LIN {X 0,Y 49.393,Z 392.721,A -85,B 0,C 180,E1 -29233.467,E2 -29233.467} C_VEL
LIN {X 0,Y 48.486,Z 393.321,A -85,B 0,C 180,E1 -29241.666,E2 -29241.666} C_VEL
LIN {X 0,Y 48.375,Z 393.484,A -85,B 0,C 180,E1 -29250,E2 -29250} C_VEL
LIN {X 0,Y 48.435,Z 393.32,A -85,B 0,C 180,E1 -29258.343,E2 -29258.343} C_VEL
LIN {X 0,Y 49.37,Z 392.721,A -85,B 0,C 180,E1 -29266.541,E2 -29266.541} C_VEL
LIN {X 0,Y 53.735,Z 390.255,A -85,B 0,C 180,E1 -29281.544,E2 -29281.544} C_VEL
LIN {X 0,Y 59.085,Z 387.3,A -85,B 0,C 180,E1 -29290.859,E2 -29290.859} C_VEL
LIN {X 0,Y 65.668,Z 383.308,A -85,B 0,C 180,E1 -29298.517,E2 -29298.517} C_VEL
LIN {X 0,Y 72.453,Z 378.717,A -85,B 0,C 180,E1 -29304.177,E2 -29304.177} C_VEL
LIN {X 0,Y 79.944,Z 372.914,A -85,B 0,C 180,E1 -29308.995,E2 -29308.995} C_VEL
LIN {X 0,Y 87.112,Z 366.6,A -85,B 0,C 180,E1 -29312.553,E2 -29312.553} C_VEL
LIN {X 0,Y 93.069,Z 360.653,A -85,B 0,C 180,E1 -29314.98,E2 -29314.98} C_VEL
LIN {X 0,Y 99.196,Z 353.732,A -85,B 0,C 180,E1 -29317.078,E2 -29317.078} C_VEL
LIN {X 0,Y 105.443,Z 345.56,A -85,B 0,C 180,E1 -29318.927,E2 -29318.927} C_VEL
LIN {X 0,Y 111.015,Z 337.057,A -85,B 0,C 180,E1 -29320.335,E2 -29320.335} C_VEL
LIN {X 0,Y 115.832,Z 328.348,A -85,B 0,C 180,E1 -29321.445,E2 -29321.445} C_VEL
LIN {X 0,Y 119.661,Z 320.167,A -85,B 0,C 180,E1 -29322.239,E2 -29322.239} C_VEL
LIN {X 0,Y 123.384,Z 310.37,A -85,B 0,C 180,E1 -29322.956,E2 -29322.956} C_VEL
LIN {X 0,Y 126.435,Z 299.742,A -85,B 0,C 180,E1 -29323.562,E2 -29323.562} C_VEL
LIN {X 0,Y 128.601,Z 289.012,A -85,B 0,C 180,E1 -29323.963,E2 -29323.963} C_VEL
LIN {X 0,Y 129.115,Z 285.094,A -85,B 0,C 180,E1 -29324.205,E2 -29324.205} C_VEL
LIN {X 0,Y 127.793,Z 281.205,A -85,B 0,C 180,E1 -29327.492,E2 -29327.492} C_VEL
LIN {X 0,Y 126.772,Z 278.417,A -85,B 0,C 180,E1 -29330.626,E2 -29330.626} C_VEL
LIN {X 0,Y 126.255,Z 276.814,A -85,B 0,C 180,E1 -29332.803,E2 -29332.803} C_VEL
LIN {X 0,Y 125.625,Z 273.412,A -85,B 0,C 180,E1 -29339.998,E2 -29339.998} C_VEL
LIN {X 0,Y 126.436,Z 277.329,A -85,B 0,C 180,E1 -29348.388,E2 -29348.388} C_VEL
LIN {X 0,Y 127.729,Z 281.02,A -85,B 0,C 180,E1 -29352.713,E2 -29352.713} C_VEL
LIN {X 0,Y 128.855,Z 284.456,A -85,B 0,C 180,E1 -29355.722,E2 -29355.722} C_VEL
LIN {X 0,Y 130.302,Z 289.66,A -85,B 0,C 180,E1 -29359.084,E2 -29359.084} C_VEL
LIN {X 0,Y 131.497,Z 296.134,A -85,B 0,C 180,E1 -29362.382,E2 -29362.382} C_VEL
LIN {X 0,Y 132.087,Z 302.134,A -85,B 0,C 180,E1 -29364.77,E2 -29364.77} C_VEL
LIN {X 0,Y 132.043,Z 313.007,A -85,B 0,C 180,E1 -29368.62,E2 -29368.62} C_VEL
LIN {X 0,Y 131.934,Z 323.425,A -85,B 0,C 180,E1 -29372.808,E2 -29372.808} C_VEL
LIN {X 0,Y 132.158,Z 331.826,A -85,B 0,C 180,E1 -29376.743,E2 -29376.743} C_VEL
LIN {X 0,Y 132.814,Z 340.077,A -85,B 0,C 180,E1 -29381.14,E2 -29381.14} C_VEL
LIN {X 0,Y 134.2,Z 347.704,A -85,B 0,C 180,E1 -29385.801,E2 -29385.801} C_VEL
LIN {X 0,Y 136.544,Z 354.485,A -85,B 0,C 180,E1 -29390.536,E2 -29390.536} C_VEL
LIN {X 0,Y 139.844,Z 360.628,A -85,B 0,C 180,E1 -29395.315,E2 -29395.315} C_VEL
LIN {X 0,Y 140.999,Z 363.415,A -85,B 0,C 180,E1 -29397.416,E2 -29397.416} C_VEL
LIN {X 0,Y 142.641,Z 371.776,A -85,B 0,C 180,E1 -29403.755,E2 -29403.755} C_VEL
LIN {X 0,Y 144.297,Z 373.849,A -85,B 0,C 180,E1 -29405.827,E2 -29405.827} C_VEL
LIN {X 0,Y 145.123,Z 374.442,A -85,B 0,C 180,E1 -29406.483,E2 -29406.483} C_VEL
LIN {X 0,Y 154.851,Z 379.176,A -85,B 0,C 180,E1 -29412.377,E2 -29412.377} C_VEL
LIN {X 0,Y 167.425,Z 382.818,A -85,B 0,C 180,E1 -29417.885,E2 -29417.885} C_VEL
LIN {X 0,Y 177.687,Z 384.674,A -85,B 0,C 180,E1 -29421.414,E2 -29421.414} C_VEL
LIN {X 0,Y 193.396,Z 386.26,A -85,B 0,C 180,E1 -29425.832,E2 -29425.832} C_VEL
LIN {X 0,Y 203.873,Z 386.653,A -85,B 0,C 180,E1 -29428.545,E2 -29428.545} C_VEL
LIN {X 0,Y 208.858,Z 386.586,A -85,B 0,C 180,E1 -29430,E2 -29430} C_VEL
LIN {X 0,Y 201.727,Z 386.604,A -85,B 0,C 180,E1 -29431.997,E2 -29431.997} C_VEL
LIN {X 0,Y 190.456,Z 386.065,A -85,B 0,C 180,E1 -29434.929,E2 -29434.929} C_VEL
LIN {X 0,Y 175.7,Z 384.365,A -85,B 0,C 180,E1 -29439.207,E2 -29439.207} C_VEL
LIN {X 0,Y 165.725,Z 382.447,A -85,B 0,C 180,E1 -29442.748,E2 -29442.748} C_VEL
LIN {X 0,Y 152.591,Z 378.247,A -85,B 0,C 180,E1 -29448.808,E2 -29448.808} C_VEL
LIN {X 0,Y 145.397,Z 374.629,A -85,B 0,C 180,E1 -29453.312,E2 -29453.312} C_VEL
LIN {X 0,Y 139.313,Z 370.272,A -85,B 0,C 180,E1 -29458.184,E2 -29458.184} C_VEL
LIN {X 0,Y 134.504,Z 365.209,A -85,B 0,C 180,E1 -29463.281,E2 -29463.281} C_VEL
LIN {X 0,Y 130.286,Z 357.802,A -85,B 0,C 180,E1 -29469.769,E2 -29469.769} C_VEL
LIN {X 0,Y 128.322,Z 351.588,A -85,B 0,C 180,E1 -29474.605,E2 -29474.605} C_VEL
LIN {X 0,Y 127.289,Z 344.102,A -85,B 0,C 180,E1 -29479.646,E2 -29479.646} C_VEL
LIN {X 0,Y 127.002,Z 335.855,A -85,B 0,C 180,E1 -29484.48,E2 -29484.48} C_VEL
LIN {X 0,Y 127.336,Z 326.049,A -85,B 0,C 180,E1 -29489.371,E2 -29489.371} C_VEL
LIN {X 0,Y 127.953,Z 316.617,A -85,B 0,C 180,E1 -29493.393,E2 -29493.393} C_VEL
LIN {X 0,Y 128.554,Z 307.182,A -85,B 0,C 180,E1 -29496.91,E2 -29496.91} C_VEL
LIN {X 0,Y 128.581,Z 302.017,A -85,B 0,C 180,E1 -29499.024,E2 -29499.024} C_VEL
LIN {X 0,Y 127.927,Z 296.121,A -85,B 0,C 180,E1 -29502.001,E2 -29502.001} C_VEL
LIN {X 0,Y 127.114,Z 291.06,A -85,B 0,C 180,E1 -29505.288,E2 -29505.288} C_VEL
LIN {X 0,Y 126.156,Z 287.336,A -85,B 0,C 180,E1 -29508.555,E2 -29508.555} C_VEL
LIN {X 0,Y 125.165,Z 283.684,A -85,B 0,C 180,E1 -29513.149,E2 -29513.149} C_VEL
LIN {X 0,Y 124.737,Z 280.649,A -85,B 0,C 180,E1 -29520.002,E2 -29520.002} C_VEL
LIN {X 0,Y 125.322,Z 284.186,A -85,B 0,C 180,E1 -29527.251,E2 -29527.251} C_VEL
LIN {X 0,Y 126.347,Z 287.793,A -85,B 0,C 180,E1 -29531.533,E2 -29531.533} C_VEL
LIN {X 0,Y 126.754,Z 289.331,A -85,B 0,C 180,E1 -29532.927,E2 -29532.927} C_VEL
LIN {X 0,Y 124.047,Z 301.955,A -85,B 0,C 180,E1 -29533.415,E2 -29533.415} C_VEL
LIN {X 0,Y 119.531,Z 315.538,A -85,B 0,C 180,E1 -29534.169,E2 -29534.169} C_VEL
LIN {X 0,Y 115.432,Z 324.895,A -85,B 0,C 180,E1 -29534.865,E2 -29534.865} C_VEL
LIN {X 0,Y 110.475,Z 334.165,A -85,B 0,C 180,E1 -29535.808,E2 -29535.808} C_VEL
LIN {X 0,Y 104.743,Z 343.103,A -85,B 0,C 180,E1 -29537.035,E2 -29537.035} C_VEL
LIN {X 0,Y 98.259,Z 351.624,A -85,B 0,C 180,E1 -29538.613,E2 -29538.613} C_VEL
LIN {X 0,Y 91.875,Z 358.836,A -85,B 0,C 180,E1 -29540.438,E2 -29540.438} C_VEL
LIN {X 0,Y 85.603,Z 365.032,A -85,B 0,C 180,E1 -29542.539,E2 -29542.539} C_VEL
LIN {X 0,Y 77.992,Z 371.566,A -85,B 0,C 180,E1 -29545.696,E2 -29545.696} C_VEL
LIN {X 0,Y 72.125,Z 376.067,A -85,B 0,C 180,E1 -29548.722,E2 -29548.722} C_VEL
LIN {X 0,Y 63.843,Z 381.563,A -85,B 0,C 180,E1 -29554.35,E2 -29554.35} C_VEL
LIN {X 0,Y 56.22,Z 385.889,A -85,B 0,C 180,E1 -29561.406,E2 -29561.406} C_VEL
LIN {X 0,Y 51.711,Z 388.259,A -85,B 0,C 180,E1 -29567.193,E2 -29567.193} C_VEL
LIN {X 0,Y 47.804,Z 390.063,A -85,B 0,C 180,E1 -29573.98,E2 -29573.98} C_VEL
LIN {X 0,Y 42.611,Z 392.529,A -85,B 0,C 180,E1 -29590.739,E2 -29590.739} C_VEL
LIN {X 0,Y 41.457,Z 393.129,A -85,B 0,C 180,E1 -29600.24,E2 -29600.24} C_VEL
LIN {X 0,Y 41.286,Z 393.293,A -85,B 0,C 180,E1 -29610,E2 -29610} C_VEL
LIN {X 0,Y 41.417,Z 393.128,A -85,B 0,C 180,E1 -29619.77,E2 -29619.77} C_VEL
LIN {X 0,Y 42.59,Z 392.528,A -85,B 0,C 180,E1 -29629.27,E2 -29629.27} C_VEL
LIN {X 0,Y 47.797,Z 390.062,A -85,B 0,C 180,E1 -29646.026,E2 -29646.026} C_VEL
LIN {X 0,Y 53.895,Z 387.107,A -85,B 0,C 180,E1 -29655.824,E2 -29655.824} C_VEL
LIN {X 0,Y 61.19,Z 383.116,A -85,B 0,C 180,E1 -29663.512,E2 -29663.512} C_VEL
LIN {X 0,Y 69.448,Z 377.897,A -85,B 0,C 180,E1 -29669.599,E2 -29669.599} C_VEL
LIN {X 0,Y 76.515,Z 372.722,A -85,B 0,C 180,E1 -29673.578,E2 -29673.578} C_VEL
LIN {X 0,Y 84.072,Z 366.408,A -85,B 0,C 180,E1 -29676.858,E2 -29676.858} C_VEL
LIN {X 0,Y 90.293,Z 360.461,A -85,B 0,C 180,E1 -29679.07,E2 -29679.07} C_VEL
LIN {X 0,Y 96.647,Z 353.54,A -85,B 0,C 180,E1 -29680.966,E2 -29680.966} C_VEL
LIN {X 0,Y 103.099,Z 345.368,A -85,B 0,C 180,E1 -29682.619,E2 -29682.619} C_VEL
LIN {X 0,Y 108.833,Z 336.866,A -85,B 0,C 180,E1 -29683.854,E2 -29683.854} C_VEL
LIN {X 0,Y 113.776,Z 328.157,A -85,B 0,C 180,E1 -29684.83,E2 -29684.83} C_VEL
LIN {X 0,Y 118.232,Z 318.697,A -85,B 0,C 180,E1 -29685.597,E2 -29685.597} C_VEL
LIN {X 0,Y 121.853,Z 309.038,A -85,B 0,C 180,E1 -29686.236,E2 -29686.236} C_VEL
LIN {X 0,Y 124.785,Z 298.851,A -85,B 0,C 180,E1 -29686.709,E2 -29686.709} C_VEL
LIN {X 0,Y 126.714,Z 289.278,A -85,B 0,C 180,E1 -29687.107,E2 -29687.107} C_VEL
LIN {X 0,Y 125.662,Z 285.548,A -85,B 0,C 180,E1 -29690.948,E2 -29690.948} C_VEL
LIN {X 0,Y 125.181,Z 283.624,A -85,B 0,C 180,E1 -29693.551,E2 -29693.551} C_VEL
LIN {X 0,Y 124.737,Z 280.648,A -85,B 0,C 180,E1 -29700.402,E2 -29700.402} C_VEL
LIN {X 0,Y 125.307,Z 284.348,A -85,B 0,C 180,E1 -29707.856,E2 -29707.856} C_VEL
LIN {X 0,Y 126.224,Z 287.718,A -85,B 0,C 180,E1 -29711.846,E2 -29711.846} C_VEL
LIN {X 0,Y 127.338,Z 292.134,A -85,B 0,C 180,E1 -29715.504,E2 -29715.504} C_VEL
LIN {X 0,Y 128.222,Z 298.337,A -85,B 0,C 180,E1 -29719.198,E2 -29719.198} C_VEL
LIN {X 0,Y 128.611,Z 303.69,A -85,B 0,C 180,E1 -29721.727,E2 -29721.727} C_VEL
LIN {X 0,Y 128.325,Z 312.227,A -85,B 0,C 180,E1 -29724.94,E2 -29724.94} C_VEL
LIN {X 0,Y 127.613,Z 321.968,A -85,B 0,C 180,E1 -29728.807,E2 -29728.807} C_VEL
LIN {X 0,Y 127.108,Z 330.9,A -85,B 0,C 180,E1 -29732.935,E2 -29732.935} C_VEL
LIN {X 0,Y 127.006,Z 339.387,A -85,B 0,C 180,E1 -29737.493,E2 -29737.493} C_VEL
LIN {X 0,Y 127.698,Z 347.955,A -85,B 0,C 180,E1 -29742.891,E2 -29742.891} C_VEL
LIN {X 0,Y 129.326,Z 355.257,A -85,B 0,C 180,E1 -29748.192,E2 -29748.192} C_VEL
LIN {X 0,Y 131.901,Z 361.133,A -85,B 0,C 180,E1 -29753.054,E2 -29753.054} C_VEL
LIN {X 0,Y 135.667,Z 366.605,A -85,B 0,C 180,E1 -29758.088,E2 -29758.088} C_VEL
LIN {X 0,Y 141.285,Z 371.898,A -85,B 0,C 180,E1 -29763.554,E2 -29763.554} C_VEL
LIN {X 0,Y 145.123,Z 374.442,A -85,B 0,C 180,E1 -29766.483,E2 -29766.483} C_VEL
LIN {X 0,Y 147.382,Z 376.327,A -85,B 0,C 180,E1 -29768.499,E2 -29768.499} C_VEL
LIN {X 0,Y 151.083,Z 380.668,A -85,B 0,C 180,E1 -29773.359,E2 -29773.359} C_VEL
LIN {X 0,Y 154.173,Z 382.556,A -85,B 0,C 180,E1 -29775.98,E2 -29775.98} C_VEL
LIN {X 0,Y 156.419,Z 383.205,A -85,B 0,C 180,E1 -29777.139,E2 -29777.139} C_VEL
LIN {X 0,Y 170.232,Z 385.537,A -85,B 0,C 180,E1 -29782.227,E2 -29782.227} C_VEL
LIN {X 0,Y 183.171,Z 386.644,A -85,B 0,C 180,E1 -29785.993,E2 -29785.993} C_VEL
LIN {X 0,Y 190.534,Z 386.905,A -85,B 0,C 180,E1 -29787.886,E2 -29787.886} C_VEL
LIN {X 0,Y 198.866,Z 386.851,A -85,B 0,C 180,E1 -29790,E2 -29790} C_VEL
LIN {X 0,Y 189.901,Z 386.887,A -85,B 0,C 180,E1 -29792.27,E2 -29792.27} C_VEL
LIN {X 0,Y 176.604,Z 386.208,A -85,B 0,C 180,E1 -29795.814,E2 -29795.814} C_VEL
LIN {X 0,Y 163.96,Z 384.68,A -85,B 0,C 180,E1 -29799.872,E2 -29799.872} C_VEL
LIN {X 0,Y 152.512,Z 382.193,A -85,B 0,C 180,E1 -29804.605,E2 -29804.605} C_VEL
LIN {X 0,Y 144.692,Z 379.654,A -85,B 0,C 180,E1 -29808.715,E2 -29808.715} C_VEL
LIN {X 0,Y 135.883,Z 375.063,A -85,B 0,C 180,E1 -29814.915,E2 -29814.915} C_VEL
LIN {X 0,Y 130.276,Z 370.556,A -85,B 0,C 180,E1 -29820.332,E2 -29820.332} C_VEL
LIN {X 0,Y 125.489,Z 364.128,A -85,B 0,C 180,E1 -29827.057,E2 -29827.057} C_VEL
LIN {X 0,Y 123.198,Z 358.678,A -85,B 0,C 180,E1 -29832.135,E2 -29832.135} C_VEL
LIN {X 0,Y 121.925,Z 352.101,A -85,B 0,C 180,E1 -29837.478,E2 -29837.478} C_VEL
LIN {X 0,Y 121.545,Z 343.222,A -85,B 0,C 180,E1 -29843.657,E2 -29843.657} C_VEL
LIN {X 0,Y 122.109,Z 335.594,A -85,B 0,C 180,E1 -29848.132,E2 -29848.132} C_VEL
LIN {X 0,Y 123.177,Z 326.23,A -85,B 0,C 180,E1 -29852.844,E2 -29852.844} C_VEL
LIN {X 0,Y 124.406,Z 317.146,A -85,B 0,C 180,E1 -29856.708,E2 -29856.708} C_VEL
LIN {X 0,Y 125.31,Z 308.99,A -85,B 0,C 180,E1 -29859.939,E2 -29859.939} C_VEL
LIN {X 0,Y 125.375,Z 303.108,A -85,B 0,C 180,E1 -29862.804,E2 -29862.804} C_VEL
LIN {X 0,Y 124.939,Z 297.563,A -85,B 0,C 180,E1 -29866.274,E2 -29866.274} C_VEL
LIN {X 0,Y 124.395,Z 293.815,A -85,B 0,C 180,E1 -29869.627,E2 -29869.627} C_VEL
LIN {X 0,Y 123.855,Z 290.479,A -85,B 0,C 180,E1 -29873.894,E2 -29873.894} C_VEL
LIN {X 0,Y 123.667,Z 287.874,A -85,B 0,C 180,E1 -29880.002,E2 -29880.002} C_VEL
LIN {X 0,Y 123.989,Z 290.973,A -85,B 0,C 180,E1 -29886.511,E2 -29886.511} C_VEL
LIN {X 0,Y 124.523,Z 293.718,A -85,B 0,C 180,E1 -29889.862,E2 -29889.862} C_VEL
LIN {X 0,Y 121.448,Z 305.563,A -85,B 0,C 180,E1 -29890.342,E2 -29890.342} C_VEL
LIN {X 0,Y 117.656,Z 316.147,A -85,B 0,C 180,E1 -29890.869,E2 -29890.869} C_VEL
LIN {X 0,Y 113.815,Z 324.703,A -85,B 0,C 180,E1 -29891.403,E2 -29891.403} C_VEL
LIN {X 0,Y 108.757,Z 333.973,A -85,B 0,C 180,E1 -29892.208,E2 -29892.208} C_VEL
LIN {X 0,Y 102.89,Z 342.912,A -85,B 0,C 180,E1 -29893.258,E2 -29893.258} C_VEL
LIN {X 0,Y 96.227,Z 351.432,A -85,B 0,C 180,E1 -29894.599,E2 -29894.599} C_VEL
LIN {X 0,Y 89.644,Z 358.645,A -85,B 0,C 180,E1 -29896.183,E2 -29896.183} C_VEL
LIN {X 0,Y 83.132,Z 364.84,A -85,B 0,C 180,E1 -29897.998,E2 -29897.998} C_VEL
LIN {X 0,Y 75.181,Z 371.374,A -85,B 0,C 180,E1 -29900.805,E2 -29900.805} C_VEL
LIN {X 0,Y 66.93,Z 377.169,A -85,B 0,C 180,E1 -29904.554,E2 -29904.554} C_VEL
LIN {X 0,Y 60.104,Z 381.37,A -85,B 0,C 180,E1 -29908.721,E2 -29908.721} C_VEL
LIN {X 0,Y 51.768,Z 385.696,A -85,B 0,C 180,E1 -29915.457,E2 -29915.457} C_VEL
LIN {X 0,Y 46.725,Z 388.067,A -85,B 0,C 180,E1 -29921.232,E2 -29921.232} C_VEL
LIN {X 0,Y 42.24,Z 389.87,A -85,B 0,C 180,E1 -29928.278,E2 -29928.278} C_VEL
LIN {X 0,Y 35.97,Z 392.337,A -85,B 0,C 180,E1 -29946.998,E2 -29946.998} C_VEL
LIN {X 0,Y 34.477,Z 392.937,A -85,B 0,C 180,E1 -29958.238,E2 -29958.238} C_VEL
LIN {X 0,Y 34.174,Z 393.101,A -85,B 0,C 180,E1 -29970,E2 -29970} C_VEL
LIN {X 0,Y 34.419,Z 392.936,A -85,B 0,C 180,E1 -29981.782,E2 -29981.782} C_VEL
LIN {X 0,Y 35.952,Z 392.336,A -85,B 0,C 180,E1 -29993.014,E2 -29993.014} C_VEL
LIN {X 0,Y 42.235,Z 389.87,A -85,B 0,C 180,E1 -30011.729,E2 -30011.729} C_VEL
LIN {X 0,Y 49.194,Z 386.915,A -85,B 0,C 180,E1 -30021.789,E2 -30021.789} C_VEL
LIN {X 0,Y 57.246,Z 382.924,A -85,B 0,C 180,E1 -30029.246,E2 -30029.246} C_VEL
LIN {X 0,Y 66.234,Z 377.63,A -85,B 0,C 180,E1 -30035.014,E2 -30035.014} C_VEL
LIN {X 0,Y 73.618,Z 372.529,A -85,B 0,C 180,E1 -30038.556,E2 -30038.556} C_VEL
LIN {X 0,Y 81.533,Z 366.216,A -85,B 0,C 180,E1 -30041.472,E2 -30041.472} C_VEL
LIN {X 0,Y 88.007,Z 360.27,A -85,B 0,C 180,E1 -30043.39,E2 -30043.39} C_VEL
LIN {X 0,Y 94.565,Z 353.348,A -85,B 0,C 180,E1 -30045.047,E2 -30045.047} C_VEL
LIN {X 0,Y 101.206,Z 345.177,A -85,B 0,C 180,E1 -30046.454,E2 -30046.454} C_VEL
LIN {X 0,Y 107.078,Z 336.674,A -85,B 0,C 180,E1 -30047.501,E2 -30047.501} C_VEL
LIN {X 0,Y 112.128,Z 327.965,A -85,B 0,C 180,E1 -30048.333,E2 -30048.333} C_VEL
LIN {X 0,Y 116.466,Z 318.988,A -85,B 0,C 180,E1 -30048.946,E2 -30048.946} C_VEL
LIN {X 0,Y 120.361,Z 308.846,A -85,B 0,C 180,E1 -30049.523,E2 -30049.523} C_VEL
LIN {X 0,Y 123.404,Z 298.443,A -85,B 0,C 180,E1 -30049.914,E2 -30049.914} C_VEL
LIN {X 0,Y 124.518,Z 293.74,A -85,B 0,C 180,E1 -30050.137,E2 -30050.137} C_VEL
LIN {X 0,Y 123.904,Z 290.511,A -85,B 0,C 180,E1 -30054.097,E2 -30054.097} C_VEL
LIN {X 0,Y 123.628,Z 287.858,A -85,B 0,C 180,E1 -30059.998,E2 -30059.998} C_VEL
LIN {X 0,Y 123.946,Z 290.997,A -85,B 0,C 180,E1 -30066.919,E2 -30066.919} C_VEL
LIN {X 0,Y 124.458,Z 294.192,A -85,B 0,C 180,E1 -30070.779,E2 -30070.779} C_VEL
LIN {X 0,Y 125.001,Z 298.151,A -85,B 0,C 180,E1 -30074.134,E2 -30074.134} C_VEL
LIN {X 0,Y 125.395,Z 303.947,A -85,B 0,C 180,E1 -30077.676,E2 -30077.676} C_VEL
LIN {X 0,Y 125.278,Z 309.947,A -85,B 0,C 180,E1 -30080.463,E2 -30080.463} C_VEL
LIN {X 0,Y 123.776,Z 321.881,A -85,B 0,C 180,E1 -30085.201,E2 -30085.201} C_VEL
LIN {X 0,Y 122.516,Z 331.392,A -85,B 0,C 180,E1 -30089.616,E2 -30089.616} C_VEL
LIN {X 0,Y 121.73,Z 340.412,A -85,B 0,C 180,E1 -30094.646,E2 -30094.646} C_VEL
LIN {X 0,Y 121.567,Z 347.926,A -85,B 0,C 180,E1 -30099.486,E2 -30099.486} C_VEL
LIN {X 0,Y 122.37,Z 355.535,A -85,B 0,C 180,E1 -30105.224,E2 -30105.224} C_VEL
LIN {X 0,Y 124.287,Z 361.676,A -85,B 0,C 180,E1 -30110.588,E2 -30110.588} C_VEL
LIN {X 0,Y 127.787,Z 367.773,A -85,B 0,C 180,E1 -30116.635,E2 -30116.635} C_VEL
LIN {X 0,Y 133.763,Z 373.584,A -85,B 0,C 180,E1 -30123.273,E2 -30123.273} C_VEL
LIN {X 0,Y 139.961,Z 377.442,A -85,B 0,C 180,E1 -30128.233,E2 -30128.233} C_VEL
LIN {X 0,Y 148.703,Z 381.049,A -85,B 0,C 180,E1 -30133.527,E2 -30133.527} C_VEL
LIN {X 0,Y 156.419,Z 383.205,A -85,B 0,C 180,E1 -30137.139,E2 -30137.139} C_VEL
LIN {X 0,Y 159.788,Z 384.124,A -85,B 0,C 180,E1 -30138.869,E2 -30138.869} C_VEL
LIN {X 0,Y 164.289,Z 385.698,A -85,B 0,C 180,E1 -30141.948,E2 -30141.948} C_VEL
LIN {X 0,Y 169.272,Z 386.785,A -85,B 0,C 180,E1 -30144.857,E2 -30144.857} C_VEL
LIN {X 0,Y 173.282,Z 387.036,A -85,B 0,C 180,E1 -30146.295,E2 -30146.295} C_VEL
LIN {X 0,Y 182.767,Z 387.253,A -85,B 0,C 180,E1 -30148.75,E2 -30148.75} C_VEL
LIN {X 0,Y 187.774,Z 387.145,A -85,B 0,C 180,E1 -30150,E2 -30150} C_VEL
LIN {X 0,Y 175.934,Z 387.132,A -85,B 0,C 180,E1 -30152.984,E2 -30152.984} C_VEL
LIN {X 0,Y 160.739,Z 386.109,A -85,B 0,C 180,E1 -30157.537,E2 -30157.537} C_VEL
LIN {X 0,Y 150.573,Z 384.607,A -85,B 0,C 180,E1 -30161.436,E2 -30161.436} C_VEL
LIN {X 0,Y 144.891,Z 383.432,A -85,B 0,C 180,E1 -30164.052,E2 -30164.052} C_VEL
LIN {X 0,Y 134.643,Z 380.067,A -85,B 0,C 180,E1 -30170.029,E2 -30170.029} C_VEL
LIN {X 0,Y 126.26,Z 375.254,A -85,B 0,C 180,E1 -30177.054,E2 -30177.054} C_VEL
LIN {X 0,Y 121.412,Z 370.656,A -85,B 0,C 180,E1 -30182.972,E2 -30182.972} C_VEL
LIN {X 0,Y 118.032,Z 365.059,A -85,B 0,C 180,E1 -30189.283,E2 -30189.283} C_VEL
LIN {X 0,Y 116.156,Z 358.361,A -85,B 0,C 180,E1 -30195.819,E2 -30195.819} C_VEL
LIN {X 0,Y 115.842,Z 350.768,A -85,B 0,C 180,E1 -30202.063,E2 -30202.063} C_VEL
LIN {X 0,Y 116.478,Z 343.577,A -85,B 0,C 180,E1 -30207.112,E2 -30207.112} C_VEL
LIN {X 0,Y 117.623,Z 336.409,A -85,B 0,C 180,E1 -30211.447,E2 -30211.447} C_VEL
LIN {X 0,Y 119.368,Z 327.269,A -85,B 0,C 180,E1 -30216.125,E2 -30216.125} C_VEL
LIN {X 0,Y 121.239,Z 317.864,A -85,B 0,C 180,E1 -30220.168,E2 -30220.168} C_VEL
LIN {X 0,Y 122.29,Z 311.483,A -85,B 0,C 180,E1 -30222.9,E2 -30222.9} C_VEL
LIN {X 0,Y 122.492,Z 306.156,A -85,B 0,C 180,E1 -30225.888,E2 -30225.888} C_VEL
LIN {X 0,Y 122.529,Z 302.67,A -85,B 0,C 180,E1 -30228.419,E2 -30228.419} C_VEL
LIN {X 0,Y 122.296,Z 299.251,A -85,B 0,C 180,E1 -30231.742,E2 -30231.742} C_VEL
LIN {X 0,Y 122.095,Z 297.012,A -85,B 0,C 180,E1 -30235.049,E2 -30235.049} C_VEL
LIN {X 0,Y 122.218,Z 294.995,A -85,B 0,C 180,E1 -30240.002,E2 -30240.002} C_VEL
LIN {X 0,Y 122.258,Z 297.827,A -85,B 0,C 180,E1 -30245.982,E2 -30245.982} C_VEL
LIN {X 0,Y 122.307,Z 298.418,A -85,B 0,C 180,E1 -30246.769,E2 -30246.769} C_VEL
LIN {X 0,Y 119.281,Z 308.654,A -85,B 0,C 180,E1 -30247.145,E2 -30247.145} C_VEL
LIN {X 0,Y 115.07,Z 319.369,A -85,B 0,C 180,E1 -30247.614,E2 -30247.614} C_VEL
LIN {X 0,Y 109.192,Z 331.013,A -85,B 0,C 180,E1 -30248.28,E2 -30248.28} C_VEL
LIN {X 0,Y 102.349,Z 341.586,A -85,B 0,C 180,E1 -30249.22,E2 -30249.22} C_VEL
LIN {X 0,Y 96.383,Z 349.323,A -85,B 0,C 180,E1 -30250.144,E2 -30250.144} C_VEL
LIN {X 0,Y 87.929,Z 358.453,A -85,B 0,C 180,E1 -30251.732,E2 -30251.732} C_VEL
LIN {X 0,Y 81.218,Z 364.648,A -85,B 0,C 180,E1 -30253.224,E2 -30253.224} C_VEL
LIN {X 0,Y 72.955,Z 371.182,A -85,B 0,C 180,E1 -30255.565,E2 -30255.565} C_VEL
LIN {X 0,Y 66.448,Z 375.681,A -85,B 0,C 180,E1 -30257.846,E2 -30257.846} C_VEL
LIN {X 0,Y 57.018,Z 381.177,A -85,B 0,C 180,E1 -30262.416,E2 -30262.416} C_VEL
LIN {X 0,Y 47.976,Z 385.503,A -85,B 0,C 180,E1 -30268.487,E2 -30268.487} C_VEL
LIN {X 0,Y 42.365,Z 387.874,A -85,B 0,C 180,E1 -30273.959,E2 -30273.959} C_VEL
LIN {X 0,Y 37.218,Z 389.677,A -85,B 0,C 180,E1 -30280.945,E2 -30280.945} C_VEL
LIN {X 0,Y 29.531,Z 392.144,A -85,B 0,C 180,E1 -30301.578,E2 -30301.578} C_VEL
LIN {X 0,Y 27.546,Z 392.745,A -85,B 0,C 180,E1 -30315.218,E2 -30315.218} C_VEL
LIN {X 0,Y 27.064,Z 392.909,A -85,B 0,C 180,E1 -30330,E2 -30330} C_VEL
LIN {X 0,Y 27.499,Z 392.744,A -85,B 0,C 180,E1 -30344.807,E2 -30344.807} C_VEL
LIN {X 0,Y 29.516,Z 392.144,A -85,B 0,C 180,E1 -30358.438,E2 -30358.438} C_VEL
LIN {X 0,Y 37.213,Z 389.677,A -85,B 0,C 180,E1 -30379.062,E2 -30379.062} C_VEL
LIN {X 0,Y 45.134,Z 386.722,A -85,B 0,C 180,E1 -30388.917,E2 -30388.917} C_VEL
LIN {X 0,Y 53.955,Z 382.732,A -85,B 0,C 180,E1 -30395.753,E2 -30395.753} C_VEL
LIN {X 0,Y 61.866,Z 378.46,A -85,B 0,C 180,E1 -30400.071,E2 -30400.071} C_VEL
LIN {X 0,Y 69.697,Z 373.493,A -85,B 0,C 180,E1 -30403.323,E2 -30403.323} C_VEL
LIN {X 0,Y 77.902,Z 367.399,A -85,B 0,C 180,E1 -30405.887,E2 -30405.887} C_VEL
LIN {X 0,Y 84.562,Z 361.703,A -85,B 0,C 180,E1 -30407.564,E2 -30407.564} C_VEL
LIN {X 0,Y 92.983,Z 353.156,A -85,B 0,C 180,E1 -30409.289,E2 -30409.289} C_VEL
LIN {X 0,Y 99.78,Z 344.985,A -85,B 0,C 180,E1 -30410.428,E2 -30410.428} C_VEL
LIN {X 0,Y 105.77,Z 336.483,A -85,B 0,C 180,E1 -30411.255,E2 -30411.255} C_VEL
LIN {X 0,Y 110.911,Z 327.774,A -85,B 0,C 180,E1 -30411.926,E2 -30411.926} C_VEL
LIN {X 0,Y 115.571,Z 318.186,A -85,B 0,C 180,E1 -30412.458,E2 -30412.458} C_VEL
LIN {X 0,Y 119.21,Z 308.843,A -85,B 0,C 180,E1 -30412.875,E2 -30412.875} C_VEL
LIN {X 0,Y 122.3,Z 298.439,A -85,B 0,C 180,E1 -30413.238,E2 -30413.238} C_VEL
LIN {X 0,Y 122.161,Z 297.006,A -85,B 0,C 180,E1 -30415.461,E2 -30415.461} C_VEL
LIN {X 0,Y 122.221,Z 294.969,A -85,B 0,C 180,E1 -30420.41,E2 -30420.41} C_VEL
LIN {X 0,Y 122.151,Z 297.737,A -85,B 0,C 180,E1 -30426.191,E2 -30426.191} C_VEL
LIN {X 0,Y 122.452,Z 300.765,A -85,B 0,C 180,E1 -30429.913,E2 -30429.913} C_VEL
LIN {X 0,Y 122.523,Z 304.859,A -85,B 0,C 180,E1 -30433.262,E2 -30433.262} C_VEL
LIN {X 0,Y 122.35,Z 310.685,A -85,B 0,C 180,E1 -30436.689,E2 -30436.689} C_VEL
LIN {X 0,Y 121.48,Z 316.482,A -85,B 0,C 180,E1 -30439.284,E2 -30439.284} C_VEL
LIN {X 0,Y 119.792,Z 325.049,A -85,B 0,C 180,E1 -30442.869,E2 -30442.869} C_VEL
LIN {X 0,Y 118.141,Z 333.261,A -85,B 0,C 180,E1 -30446.835,E2 -30446.835} C_VEL
LIN {X 0,Y 116.74,Z 341.627,A -85,B 0,C 180,E1 -30451.659,E2 -30451.659} C_VEL
LIN {X 0,Y 115.974,Z 348.508,A -85,B 0,C 180,E1 -30456.27,E2 -30456.27} C_VEL
LIN {X 0,Y 115.88,Z 355.668,A -85,B 0,C 180,E1 -30461.844,E2 -30461.844} C_VEL
LIN {X 0,Y 116.907,Z 361.94,A -85,B 0,C 180,E1 -30467.549,E2 -30467.549} C_VEL
LIN {X 0,Y 119.565,Z 368.043,A -85,B 0,C 180,E1 -30474,E2 -30474} C_VEL
LIN {X 0,Y 124.501,Z 373.798,A -85,B 0,C 180,E1 -30481.037,E2 -30481.037} C_VEL
LIN {X 0,Y 130.202,Z 377.784,A -85,B 0,C 180,E1 -30486.576,E2 -30486.576} C_VEL
LIN {X 0,Y 138.085,Z 381.342,A -85,B 0,C 180,E1 -30492.219,E2 -30492.219} C_VEL
LIN {X 0,Y 144.92,Z 383.441,A -85,B 0,C 180,E1 -30495.967,E2 -30495.967} C_VEL
LIN {X 0,Y 156.567,Z 385.631,A -85,B 0,C 180,E1 -30500.935,E2 -30500.935} C_VEL
LIN {X 0,Y 173.282,Z 387.036,A -85,B 0,C 180,E1 -30506.295,E2 -30506.295} C_VEL
LIN {X 0,Y 174.464,Z 387.172,A -85,B 0,C 180,E1 -30506.977,E2 -30506.977} C_VEL
LIN {X 0,Y 174.49,Z 387.419,A -85,B 0,C 180,E1 -30508.079,E2 -30508.079} C_VEL
LIN {X 0,Y 172.876,Z 387.563,A -85,B 0,C 180,E1 -30509.523,E2 -30509.523} C_VEL
LIN {X 0,Y 170.764,Z 387.595,A -85,B 0,C 180,E1 -30510.586,E2 -30510.586} C_VEL
LIN {X 0,Y 167.521,Z 387.632,A -85,B 0,C 180,E1 -30511.822,E2 -30511.822} C_VEL
LIN {X 0,Y 160.497,Z 387.37,A -85,B 0,C 180,E1 -30514.198,E2 -30514.198} C_VEL
LIN {X 0,Y 156.857,Z 387.171,A -85,B 0,C 180,E1 -30515.379,E2 -30515.379} C_VEL
LIN {X 0,Y 141.237,Z 385.292,A -85,B 0,C 180,E1 -30521.481,E2 -30521.481} C_VEL
LIN {X 0,Y 131.914,Z 383.111,A -85,B 0,C 180,E1 -30526.473,E2 -30526.473} C_VEL
LIN {X 0,Y 122.603,Z 379.244,A -85,B 0,C 180,E1 -30533.489,E2 -30533.489} C_VEL
LIN {X 0,Y 116.638,Z 375.051,A -85,B 0,C 180,E1 -30540.03,E2 -30540.03} C_VEL
LIN {X 0,Y 112.992,Z 370.669,A -85,B 0,C 180,E1 -30546.046,E2 -30546.046} C_VEL
LIN {X 0,Y 110.533,Z 364.815,A -85,B 0,C 180,E1 -30553.018,E2 -30553.018} C_VEL
LIN {X 0,Y 109.892,Z 358.884,A -85,B 0,C 180,E1 -30559.046,E2 -30559.046} C_VEL
LIN {X 0,Y 110.323,Z 352.039,A -85,B 0,C 180,E1 -30565.019,E2 -30565.019} C_VEL
LIN {X 0,Y 112.08,Z 343.089,A -85,B 0,C 180,E1 -30571.385,E2 -30571.385} C_VEL
LIN {X 0,Y 113.886,Z 336.004,A -85,B 0,C 180,E1 -30575.636,E2 -30575.636} C_VEL
LIN {X 0,Y 116.223,Z 327.398,A -85,B 0,C 180,E1 -30579.992,E2 -30579.992} C_VEL
LIN {X 0,Y 118.659,Z 317.929,A -85,B 0,C 180,E1 -30584.104,E2 -30584.104} C_VEL
LIN {X 0,Y 119.459,Z 313.508,A -85,B 0,C 180,E1 -30586.391,E2 -30586.391} C_VEL
LIN {X 0,Y 119.884,Z 309.704,A -85,B 0,C 180,E1 -30588.914,E2 -30588.914} C_VEL
LIN {X 0,Y 120.021,Z 306.684,A -85,B 0,C 180,E1 -30591.584,E2 -30591.584} C_VEL
LIN {X 0,Y 120.095,Z 304.645,A -85,B 0,C 180,E1 -30594.172,E2 -30594.172} C_VEL
LIN {X 0,Y 120.196,Z 303.275,A -85,B 0,C 180,E1 -30596.65,E2 -30596.65} C_VEL
LIN {X 0,Y 120.442,Z 302.019,A -85,B 0,C 180,E1 -30600.002,E2 -30600.002} C_VEL
LIN {X 0,Y 120.247,Z 303.506,A -85,B 0,C 180,E1 -30603.352,E2 -30603.352} C_VEL
